       #sIntLoadUnloadOP(iStartSeqCond := (#sIntLoaderInSafePos AND #sMain.iStartSeqCond AND NOT #sIntLoadUnloadOP.sInterface.Error AND NOT "DB_LoaderShuttle2".sIntLoadUnloadOP.sInterface.SequenceRun AND #sIntLoadUnloadOP.sInterface.StartRequest AND #sShuttlePosInt),
                         iJobReq := #sIntLoadUnloadOP.sInterface.StartRequest,
                         iShuttleIntLoadUnloadPos := #tAxis_U_Position.IntLoadUnload,
                         iShuttleIntLoadUnloadPosSetPoint := "DB_AxisPosMachinePLC".Axis_U1.IntLoadUnload,
                         iShuttleIntLoadUnloadOP_Pos:=#tAxis_U_Position.IntLoadUnloadOP,
                         iShuttleIntLoadUnloadOP_PosSetPoint:="DB_AxisPosMachinePLC".Axis_U1.IntLoadUnloadOP,
                         iAxisV_LoadUnloadShuttlePos := #tAxis_V_Position.LoadUnload,
                         iAxisV_LoadUnloadShuttlePosSetPoint := "DB_AxisPosMachinePLC".Axis_V.Shuttle_1.LoadUnload,
                         iAxisV_SafePos := #tAxis_V_Position.Safe,
                         iAxisV_SafePosSetPoint := "DB_AxisPosMachinePLC".Axis_V.Safe,
                         iAxisW_SafePos := #tAxis_W_Position.Safe,
                         iAxisW_SafePosSetPoint := "DB_AxisPosMachinePLC".Axis_W.Safe,
                         iAxisW_ApproachLoadUnloadPos := #tAxis_W_Position.Approach,
                         iAxisW_ApproachLoadUnloadSetPoint := "DB_AxisPosMachinePLC".Axis_W.Shuttle_1.Approach,
                         iAxisW_LoadUnloadPos := #tAxis_W_Position.LoadUnload,
                         iAxisW_LoadUnloadPosSetPoint := "DB_AxisPosMachinePLC".Axis_W.Shuttle_1.LoadUnload,
                         iShuttleMoving := #iShuttleMoving,
                         iShuttleInPos := #iShuttleInPos,
                         iAxisV_Moving := #iAxisV_Moving,
                         iAxisV_InPos := #iAxisV_InPos,
                         iAxisW_Moving := #iAxisW_Moving,
                         iAxisW_InPos := #iAxisW_InPos,
                         iDrilledPartToUnload := "DB_PartManagement".sPosition.sGripper.Drilled.Presence.Part,
                         iUnDrilledPartToLoad := "DB_PartManagement".sPosition.sShuttle1.Undrilled.Presence.Part,
                         iLoadGripperClosed := #sIntLoadUnloadOP.iLoadGripperClosed,
                         iUnloadGripperOpen := "DB_GestionGripper".sDrilledGripper.oStateOpen,
                         iPLC_DateAndTime := "DB_ReadDateAndTime".sDateAndTime,
                         iStepPause := #sIntLoadUnloadOP.iStepPause,        
                         oShuttleStartReq => #sIntLoadUnloadOP.oShuttleStartReq,
                         oShuttlePosSetPoint => #sIntLoadUnloadOP.oShuttlePosSetPoint,
                         oAxisV_StartReq => #sIntLoadUnloadOP.oAxisV_StartReq,
                         oAxisV_PosSetPoint => #sIntLoadUnloadOP.oAxisV_PosSetPoint,
                         oAxisW_StartReq => #sIntLoadUnloadOP.oAxisW_StartReq,
                         oAxisW_PosSetPoint => #sIntLoadUnloadOP.oAxisW_PosSetPoint,
                         oLoadGripperCloseReq => #sIntLoadUnloadOP.oLoadGripperCloseReq,
                         oUnloadGripperOpenReq => #sIntLoadUnloadOP.oUnloadGripperOpenReq);
   END_REGION

   REGION Parts Control
       // Control In

       // Expected control result
      IF "DB_WorkingModes".sFilling THEN
          #sControlIn.iExpectedCtrlUndrilled := TRUE;
          #sControlIn.iExpectedCtrlDrilled := FALSE;
      ELSIF "DB_WorkingModes".sNormal THEN
          #sControlIn.iExpectedCtrlUndrilled := TRUE;
          #sControlIn.iExpectedCtrlDrilled := FALSE;
      ELSIF "DB_WorkingModes".sEmptying THEN
          #sControlIn.iExpectedCtrlUndrilled := FALSE;
          #sControlIn.iExpectedCtrlDrilled := FALSE;
      END_IF;

       #sControlIn(iStartSeqCond := (#sExtLoaderInSafePos AND #sMain.iStartSeqCond AND NOT #sControlIn.sInterface.Error AND NOT "DB_LoaderShuttle2".sControlIn.sInterface.SequenceRun AND #sControlIn.sInterface.StartRequest AND #sShuttlePosExt),
                   iJobReq := #sControlIn.sInterface.StartRequest,
                   iCtrlEnabled := TRUE,
                   iShuttleCtrlPos:= #tAxis_U_Position.PartControl,
                   iShuttleCtrlPosSetPoint:="DB_AxisPosMachinePLC".Axis_U1.PartControl,
                   iExpectedCtrlUndrilled := #sControlIn.iExpectedCtrlUndrilled,
                   iExpectedCtrlDrilled := #sControlIn.iExpectedCtrlDrilled,
                   iUndrilledPartPresence:= "DB_DigitalInputsBW_Station".sUndrilledPartCtrl.sSWStatus,
                   iDrilledPartPresence:= "DB_DigitalInputsBW_Station".sDrilledPartCtrl.sSWStatus,
                   iShuttleMoving := #iShuttleMoving,
                   iShuttleInPos := #iShuttleInPos,
                   iPLC_DateAndTime:= "DB_ReadDateAndTime".sDateAndTime,
                   iStepPause:=#sControlIn.iStepPause,       
                   oShuttleStartReq => #sControlIn.oShuttleStartReq,
                   oShuttlePosSetPoint => #sControlIn.oShuttlePosSetPoint,
                   oPartControlOK => #sControlIn.oPartControlOK,
                   oPartControlNOK => #sControlIn.oPartControlNOK);

       // Control Out

       // Expected control result
       #sControlOut.iExpectedCtrlUndrilled := "DB_PartManagement".sPosition.sShuttle1.Undrilled.Presence.Part;
       #sControlOut.iExpectedCtrlDrilled := "DB_PartManagement".sPosition.sShuttle1.Drilled.Presence.Part;

       #sControlOut(iStartSeqCond := (#sBwLoaderInSafePos AND #sMain.iStartSeqCond AND NOT #sControlOut.sInterface.Error AND NOT "DB_LoaderShuttle2".sControlOut.sInterface.SequenceRun AND #sControlOut.sInterface.StartRequest AND #sShuttlePosExt),
                    iJobReq := #sControlOut.sInterface.StartRequest,
                    iCtrlEnabled := TRUE,
                    iShuttleCtrlPos:= #tAxis_U_Position.PartControl,
                    iShuttleCtrlPosSetPoint:= "DB_AxisPosMachinePLC".Axis_U1.PartControl,
                    iExpectedCtrlUndrilled := #sControlOut.iExpectedCtrlUndrilled,
                    iExpectedCtrlDrilled := #sControlOut.iExpectedCtrlDrilled,
                    iUndrilledPartPresence:="DB_DigitalInputsBW_Station".sUndrilledPartCtrl.sSWStatus,
                    iDrilledPartPresence:="DB_DigitalInputsBW_Station".sDrilledPartCtrl.sSWStatus,
                    iShuttleMoving := #iShuttleMoving,
                    iShuttleInPos := #iShuttleInPos,
                    iPLC_DateAndTime:= "DB_ReadDateAndTime".sDateAndTime,
                    iStepPause:=#sControlOut.iStepPause,     
                    oShuttleStartReq => #sControlOut.oShuttleStartReq,
                    oShuttlePosSetPoint => #sControlOut.oShuttlePosSetPoint,
                    oPartControlOK => #sControlOut.oPartControlOK,
                    oPartControlNOK => #sControlOut.oPartControlNOK);
   END_REGION

   REGION BW Load Unload
       #sBwLoadUnload(iStartSeqCond:= (#sMain.iStartSeqCond AND NOT #sBwLoadUnload.sInterface.Error AND NOT "DB_LoaderShuttle2".sBwLoadUnload.sInterface.SequenceRun AND #sBwLoadUnload.sInterface.StartRequest AND #sShuttlePosExt),
                      iJobReq:= #sBwLoadUnload.sInterface.StartRequest,
                      iLoadReq:= #sMain.oBwLoadReq,
                      iUnloadReq:= #sMain.oBwUnloadReq,
                      iShuttleBwUnloadPos:= #tAxis_U_Position.BwUnload,
                      iShuttleBwUnloadPosSetPoint:= "DB_AxisPosMachinePLC".Axis_U1.BwUnLoad,
                      iShuttleBwLoadPos:= #tAxis_U_Position.BwLoad,
                      iShuttleBwLoadPosSetPoint:= "DB_AxisPosMachinePLC".Axis_U1.BwLoad,
                      iShuttleMoving:= #iShuttleMoving,
                      iShuttleInPos:= #iShuttleInPos,
                      iBwLoadDone:="DB_BwLoader".sBwCommunication.oLoadJobDone,
                      iBwUnloadDone:="DB_BwLoader".sBwCommunication.oUnloadJobDone,
                      iBwLoaderInSafePos:=#sBwLoaderInSafePos,
                      iPLC_DateAndTime:= "DB_ReadDateAndTime".sDateAndTime,
                      iStepPause:=#sBwLoadUnload.iStepPause,      
                      oShuttleStartReq=> #sBwLoadUnload.oShuttleStartReq,
                      oShuttlePosSetPoint=> #sBwLoadUnload.oShuttlePosSetPoint,
                      oBwLoadReq=> #sBwLoadUnload.oBwLoadReq,
                      oBwUnloadReq=>#sBwLoadUnload.oBwUnloadReq);
   END_REGION

   REGION BW Control
       // BW Control In

       // Expected control result
       #sBwControlIn.iExpectedCtrl := "DB_PartManagement".sPosition.sShuttle1.Undrilled.Presence.Part;

       #sBwControlIn(iStartSeqCond := (#sMain.iStartSeqCond AND NOT #sBwControlIn.sInterface.Error AND NOT "DB_LoaderShuttle2".sBwControlIn.sInterface.SequenceRun AND #sBwControlIn.sInterface.StartRequest AND #sShuttlePosExt),
                     iJobReq := #sBwControlIn.sInterface.StartRequest,
                     iCtrlEnabled := TRUE,
                     iShuttleCtrlPos := #tAxis_U_Position.BwControl,
                     iShuttleCtrlPosSetPoint := "DB_AxisPosMachinePLC".Axis_U1.BwControl,
                     iExpectedCtrl := #sBwControlIn.iExpectedCtrl,
                     iBwPresence := "DB_DigitalInputsBW_Station".sBwCtrl.sSWStatus,
                     iShuttleMoving := #iShuttleMoving,
                     iShuttleInPos := #iShuttleInPos,
                     iPLC_DateAndTime := "DB_ReadDateAndTime".sDateAndTime,
                     iStepPause := #sBwControlIn.iStepPause,     
                     oShuttleStartReq => #sBwControlIn.oShuttleStartReq,
                     oShuttlePosSetPoint => #sBwControlIn.oShuttlePosSetPoint,
                     oBwControlOK => #sBwControlIn.oBwControlOK,
                     oBwControlNOK => #sBwControlIn.oBwControlNOK);

       #sBwConsecutiveCtrl(iReset:=#sBwConsecutiveCtrl.oConsecutiveError AND #sActBwControlIn.sCurrent_Step_NB = 60,
                           iGoodEntry:=#sBwControlIn.oBwControlOK,
                           iBadEntry:=#sBwControlIn.oBwControlNOK,
                           iPresetValue:=3,
                           oConsecutiveError=>#sBwConsecutiveCtrl.oConsecutiveError);
   END_REGION

   REGION Blowing
       #sBlowing(iStartSeqCond:=(#sIntLoaderInSafePos AND #sMain.iStartSeqCond AND NOT #sBlowing.sInterface.Error AND NOT "DB_LoaderShuttle2".sBlowing.sInterface.SequenceRun AND #sBlowing.sInterface.StartRequest AND #sShuttlePosInt),
                 iJobReq:=#sBlowing.sInterface.StartRequest,
                 iShuttleBlowingPos:=#tAxis_U_Position.Blowing,
                 iShuttleBlowingPosSetPoint:="DB_AxisPosMachinePLC".Axis_U1.Blowing,
                 iAxisV_BlowingPos:=#tAxis_V_Position.Blowing,
                 iAxisV_BlowingPosSetPoint:="DB_AxisPosMachinePLC".Axis_V.Shuttle_1.Blowing,
                 iAxisW_SafePos:=#tAxis_W_Position.Safe,
                 iAxisW_SafePosSetPoint:="DB_AxisPosMachinePLC".Axis_W.Safe,
                 iAxisW_BlowingPos:=#tAxis_W_Position.Blowing,
                 iAxisW_BlowingPosSetPoint:="DB_AxisPosMachinePLC".Axis_W.Shuttle_1.Blowing,
                 iShuttleMoving:=#iShuttleMoving,
                 iShuttleInPos:=#iShuttleInPos,
                 iAxisV_Moving:=#iAxisV_Moving,
                 iAxisV_InPos:=#iAxisV_InPos,
                 iAxisW_Moving:=#iAxisW_Moving,
                 iAxisW_InPos:=#iAxisW_InPos,
                 iBlowingTime:=DINT_TO_TIME(REAL_TO_DINT("DB_HMISetting".BlowingSetpoint)),
                 iPLC_DateAndTime:="DB_ReadDateAndTime".sDateAndTime,
                 iStepPause:=#sBlowing.iStepPause,
                 oShuttleStartReq=>#sBlowing.oShuttleStartReq,
                 oShuttlePosSetPoint=>#sBlowing.oShuttlePosSetPoint,
                 oAxisV_StartReq=>#sBlowing.oAxisV_StartReq,
                 oAxisV_PosSetPoint=>#sBlowing.iAxisV_BlowingPosSetPoint,
                 oAxisW_StartReq=>#sBlowing.oAxisW_StartReq,
                 oAxisW_PosSetPoint=>#sBlowing.iAxisW_BlowingPosSetPoint,
                 oBlowingReq=>#sBlowing.oBlowingReq);
   END_REGION

   REGION Action Part Control In
       // Conditions d'arrêt en Mode Auto
       #sActPartControlIn.iModeAutoPosCondition :=
          ("DB_WorkingModes".sAuto AND (#sControlIn.sMissingPartCtrlUndrilled OR #sControlIn.sMissingPartCtrlDrilled) AND "DB_LoaderOptions".ActPartControlIn.Stop)
       OR ("DB_WorkingModes".sAuto AND (#sControlIn.sExtraPartCtrlUndrilled OR #sControlIn.sExtraPartCtrlDrilled) AND "DB_LoaderOptions".ActPartControlIn.Stop)
       OR ("DB_WorkingModes".sAuto AND (#sControlIn.sExtraPartCtrlUndrilled OR #sControlIn.sExtraPartCtrlDrilled) AND NOT "DB_LoaderOptions".ActPartControlIn.Stop);
       // Conditions d'arrêt en Mode Semi Auto   
       #sActPartControlIn.iModeSemiAutoPosCondition :=
          ("DB_WorkingModes".sSemiAuto AND (#sControlIn.sMissingPartCtrlUndrilled OR #sControlIn.sMissingPartCtrlDrilled) AND "DB_LoaderOptions".ActPartControlIn.Stop)
       OR ("DB_WorkingModes".sSemiAuto AND (#sControlIn.sExtraPartCtrlUndrilled OR #sControlIn.sExtraPartCtrlDrilled) AND "DB_LoaderOptions".ActPartControlIn.Stop)
       OR ("DB_WorkingModes".sSemiAuto AND (#sControlIn.sExtraPartCtrlUndrilled OR #sControlIn.sExtraPartCtrlDrilled) AND NOT "DB_LoaderOptions".ActPartControlIn.Stop);
       // Conditions pas d'arrêt
       #sActPartControlIn.iNoStopCondition :=
          ("DB_WorkingModes".sAuto AND (#sControlIn.sMissingPartCtrlUndrilled OR #sControlIn.sMissingPartCtrlDrilled) AND NOT "DB_LoaderOptions".ActPartControlIn.Stop)
       OR ("DB_WorkingModes".sSemiAuto AND (#sControlIn.sMissingPartCtrlUndrilled OR #sControlIn.sMissingPartCtrlDrilled) AND NOT "DB_LoaderOptions".ActPartControlIn.Stop);

       #sActPartControlIn(iStartSeqCond:= (#sMain.iStartSeqCond AND NOT #sActPartControlIn.sInterface.Error AND NOT "DB_LoaderShuttle2".sActPartControlIn.sInterface.SequenceRun AND #sActPartControlIn.sInterface.StartRequest AND #sShuttlePosExt),
                          iJobReq:= #sActPartControlIn.sInterface.StartRequest,
                          iShuttleModeAutoPos:= #tAxis_U_Position.ExtLoadUnloadAuto,
                          iShuttleModeAutoPosSetPoint:= "DB_AxisPosMachinePLC".Axis_U1.ExtLoadUnloadAuto,
                          iShuttleModeSemiAutoPos:= #tAxis_U_Position.ExtLoadUnloadManu,
                          iShuttleModeSemiAutoPosSetPoint:= "DB_AxisPosMachinePLC".Axis_U1.ExtLoadUnloadManu,
                          iShuttleMoving:= #iShuttleMoving,
                          iShuttleInPos:= #iShuttleInPos,
                          iModeAutoPosCondition:= #sActPartControlIn.iModeAutoPosCondition,
                          iModeSemiAutoPosCondition:= #sActPartControlIn.iModeSemiAutoPosCondition,
                          iNoStopCondition:= #sActPartControlIn.iNoStopCondition,
                          iOperatorCycleRestart:= "LBP_Chan1".E_ProgRunning,
                          iNC_Stopped:= NOT "LBP_Chan1".E_ProgRunning,
                          iNC_Running:= "LBP_Chan1".E_ProgRunning,
                          iMissingPart:=#sControlIn.sMissingPartCtrlUndrilled OR #sControlIn.sMissingPartCtrlDrilled,
                          iExtraPart:=#sControlIn.sExtraPartCtrlUndrilled OR #sControlIn.sExtraPartCtrlDrilled,
                          iPLC_DateAndTime:= "DB_ReadDateAndTime".sDateAndTime,
                          iStepPause:= #sActPartControlIn.iStepPause,
                          oShuttleStartReq=> #sActPartControlIn.oShuttleStartReq,
                          oShuttlePosSetPoint=> #sActPartControlIn.oShuttlePosSetPoint,
                          oStopNC_Req=> #sActPartControlIn.oStopNC_Req,       // Implicite par Alarm Message
                          oRestartNC_Req=> #sActPartControlIn.oRestartNC_Req, // Implicite par Restart NC
                          oRestartStep=> #sActPartControlIn.oRestartStep,
                          oContinuationStep=> #sActPartControlIn.oContinuationStep,
                          oMsgMissingPart=>#sActPartControlIn.oMsgMissingPart,
                          oMsgExtraPart=>#sActPartControlIn.oMsgExtraPart);

       #sRT_PartControlInMissing(CLK := #sActPartControlIn.oMsgMissingPart);
       IF #sRT_PartControlInMissing.Q THEN
           "LBP_AlarmMsgs".UserA[03].A70UUxx[15] := TRUE;
       END_IF;

       #sRT_PartControlInExtra(CLK := #sActPartControlIn.oMsgExtraPart);
       IF #sRT_PartControlInExtra.Q THEN
           "LBP_AlarmMsgs".UserA[03].A70UUxx[16] := TRUE;
       END_IF;
   END_REGION

   REGION Action Part Control Out
       // Conditions d'arrêt en Mode Auto
       #sActPartControlOut.iModeAutoPosCondition :=
          ("DB_WorkingModes".sAuto AND (#sControlOut.sMissingPartCtrlUndrilled OR #sControlOut.sMissingPartCtrlDrilled) AND "DB_LoaderOptions".ActPartControlOut.Stop)
       OR ("DB_WorkingModes".sAuto AND (#sControlOut.sExtraPartCtrlUndrilled OR #sControlOut.sExtraPartCtrlDrilled) AND "DB_LoaderOptions".ActPartControlOut.Stop)
       OR ("DB_WorkingModes".sAuto AND (#sControlOut.sExtraPartCtrlUndrilled OR #sControlOut.sExtraPartCtrlDrilled) AND NOT "DB_LoaderOptions".ActPartControlOut.Stop);
       // Conditions d'arrêt en Mode Semi Auto 
       #sActPartControlOut.iModeSemiAutoPosCondition :=
          ("DB_WorkingModes".sSemiAuto AND (#sControlOut.sMissingPartCtrlUndrilled OR #sControlOut.sMissingPartCtrlDrilled) AND "DB_LoaderOptions".ActPartControlOut.Stop)
       OR ("DB_WorkingModes".sSemiAuto AND (#sControlOut.sExtraPartCtrlUndrilled OR #sControlOut.sExtraPartCtrlDrilled) AND "DB_LoaderOptions".ActPartControlOut.Stop)
       OR ("DB_WorkingModes".sSemiAuto AND (#sControlOut.sExtraPartCtrlUndrilled OR #sControlOut.sExtraPartCtrlDrilled) AND NOT "DB_LoaderOptions".ActPartControlOut.Stop);
       // Conditions pas d'arrêt
       #sActPartControlOut.iNoStopCondition :=
          ("DB_WorkingModes".sAuto AND (#sControlOut.sMissingPartCtrlUndrilled OR #sControlOut.sMissingPartCtrlDrilled) AND NOT "DB_LoaderOptions".ActPartControlOut.Stop)
       OR ("DB_WorkingModes".sSemiAuto AND (#sControlOut.sMissingPartCtrlUndrilled OR #sControlOut.sMissingPartCtrlDrilled) AND NOT "DB_LoaderOptions".ActPartControlOut.Stop);

       #sActPartControlOut(iStartSeqCond := (#sMain.iStartSeqCond AND NOT #sActPartControlOut.sInterface.Error AND NOT "DB_LoaderShuttle2".sActPartControlout.sInterface.SequenceRun AND #sActPartControlOut.sInterface.StartRequest AND #sShuttlePosExt),
                           iJobReq := #sActPartControlOut.sInterface.StartRequest,
                           iShuttleModeAutoPos := #tAxis_U_Position.ExtLoadUnloadAuto,
                           iShuttleModeAutoPosSetPoint := "DB_AxisPosMachinePLC".Axis_U1.ExtLoadUnloadAuto,
                           iShuttleModeSemiAutoPos := #tAxis_U_Position.ExtLoadUnloadManu,
                           iShuttleModeSemiAutoPosSetPoint := "DB_AxisPosMachinePLC".Axis_U1.ExtLoadUnloadManu,
                           iShuttleMoving := #iShuttleMoving,
                           iShuttleInPos := #iShuttleInPos,
                           iModeAutoPosCondition := #sActPartControlOut.iModeAutoPosCondition,
                           iModeSemiAutoPosCondition := #sActPartControlOut.iModeSemiAutoPosCondition,
                           iNoStopCondition:=#sActPartControlOut.iNoStopCondition,
                           iOperatorCycleRestart := "LBP_Chan1".E_ProgRunning,
                           iNC_Stopped := NOT "LBP_Chan1".E_ProgRunning,
                           iNC_Running := "LBP_Chan1".E_ProgRunning,
                           iMissingPart:=#sControlOut.sMissingPartCtrlUndrilled OR #sControlOut.sMissingPartCtrlDrilled,
                           iExtraPart:=#sControlOut.sExtraPartCtrlUndrilled OR #sControlOut.sExtraPartCtrlDrilled,
                           iPLC_DateAndTime := "DB_ReadDateAndTime".sDateAndTime,
                           iStepPause := #sActPartControlOut.iStepPause, 
                           oShuttleStartReq => #sActPartControlOut.oShuttleStartReq,
                           oShuttlePosSetPoint => #sActPartControlOut.oShuttlePosSetPoint,
                           oStopNC_Req => #sActPartControlOut.oStopNC_Req,       // Implicite par Alarm Message
                           oRestartNC_Req => #sActPartControlOut.oRestartNC_Req, // Implicite par Restart NC
                           oRestartStep => #sActPartControlOut.oRestartStep,
                           oContinuationStep => #sActPartControlOut.oContinuationStep,
                           oMsgMissingPart=>#sActPartControlOut.oMsgMissingPart,
                           oMsgExtraPart=>#sActPartControlOut.oMsgExtraPart);

      #sRT_PartControlOutMissing(CLK := #sActPartControlOut.oMsgMissingPart);
      IF #sRT_PartControlOutMissing.Q THEN
          "LBP_AlarmMsgs".UserA[03].A70UUxx[17] := TRUE;
      END_IF;

      #sRT_PartControlOutExtra(CLK := #sActPartControlOut.oMsgExtraPart);
      IF #sRT_PartControlOutExtra.Q THEN
          "LBP_AlarmMsgs".UserA[03].A70UUxx[18] := TRUE;
      END_IF;
   END_REGION

   REGION Action Bw Control In
       // Conditions d'arrêt en Mode Auto
       #sActBwControlIn.iModeAutoPosCondition :=
       ("DB_WorkingModes".sAuto AND #sBwControlIn.sMissingBwCtrl AND ("DB_LoaderOptions".ActBwControlIn.Stop OR #sBwConsecutiveCtrl.oConsecutiveError))
       OR ("DB_WorkingModes".sAuto AND #sBwControlIn.sExtraBwCtrl AND "DB_LoaderOptions".ActBwControlIn.Stop)
       OR ("DB_WorkingModes".sAuto AND #sBwControlIn.sExtraBwCtrl AND NOT "DB_LoaderOptions".ActBwControlIn.Stop);
       // Conditions d'arrêt en Mode Semi Auto
       #sActBwControlIn.iModeSemiAutoPosCondition :=
          ("DB_WorkingModes".sSemiAuto AND #sBwControlIn.sMissingBwCtrl AND "DB_LoaderOptions".ActBwControlIn.Stop)
       OR ("DB_WorkingModes".sSemiAuto AND #sBwControlIn.sExtraBwCtrl AND "DB_LoaderOptions".ActBwControlIn.Stop)
       OR ("DB_WorkingModes".sSemiAuto AND #sBwControlIn.sExtraBwCtrl AND NOT "DB_LoaderOptions".ActBwControlIn.Stop);
       // Conditions pas d'arrêt
       #sActBwControlIn.iNoStopCondition :=
       ("DB_WorkingModes".sAuto AND #sBwControlIn.sMissingBwCtrl AND (NOT "DB_LoaderOptions".ActBwControlIn.Stop AND NOT #sBwConsecutiveCtrl.oConsecutiveError))
       OR ("DB_WorkingModes".sSemiAuto AND #sBwControlIn.sMissingBwCtrl AND NOT "DB_LoaderOptions".ActBwControlIn.Stop);

       #sActBwControlIn(iStartSeqCond := (#sMain.iStartSeqCond AND NOT #sActBwControlIn.sInterface.Error AND NOT "DB_LoaderShuttle2".sActBwControlIn.sInterface.SequenceRun AND #sActBwControlIn.sInterface.StartRequest AND #sShuttlePosExt),
                        iJobReq := #sActBwControlIn.sInterface.StartRequest,
                        iShuttleModeAutoPos := #tAxis_U_Position.BwLoad,
                        iShuttleModeAutoPosSetPoint := "DB_AxisPosMachinePLC".Axis_U1.BwLoad,
                        iShuttleModeSemiAutoPos := #tAxis_U_Position.BwLoad,
                        iShuttleModeSemiAutoPosSetPoint := "DB_AxisPosMachinePLC".Axis_U1.BwLoad,
                        iShuttleMoving := #iShuttleMoving,
                        iShuttleInPos := #iShuttleInPos,
                        iModeAutoPosCondition := #sActBwControlIn.iModeAutoPosCondition,
                        iModeSemiAutoPosCondition := #sActBwControlIn.iModeSemiAutoPosCondition,
                        iNoStopCondition:=#sActBwControlIn.iNoStopCondition,
                        iOperatorCycleRestart := "LBP_Chan1".E_ProgRunning,
                        iNC_Stopped :=  (NOT "LBP_Chan1".E_ProgRunning AND "DB_OPC_Machine".Parameters.ConsecutiveBwIn = 0) OR "DB_OPC_Machine".Parameters.ConsecutiveBwIn > 0,
                        iNC_Running := "LBP_Chan1".E_ProgRunning,
                        iMissingPart:=#sBwControlIn.sMissingBwCtrl,
                        iExtraPart:=#sBwControlIn.sExtraBwCtrl,
                        iPLC_DateAndTime := "DB_ReadDateAndTime".sDateAndTime,
                        iStepPause := #sActBwControlIn.iStepPause,
                        oShuttleStartReq => #sActBwControlIn.oShuttleStartReq,
                        oShuttlePosSetPoint => #sActBwControlIn.oShuttlePosSetPoint,
                        oStopNC_Req => #sActBwControlIn.oStopNC_Req,       // Implicite par Alarm Message
                        oRestartNC_Req => #sActBwControlIn.oRestartNC_Req, // Implicite par Restart NC
                        oRestartStep => #sActBwControlIn.oRestartStep,
                        oContinuationStep => #sActBwControlIn.oContinuationStep,
                        oMsgMissingPart=>#sActBwControlIn.oMsgMissingPart,
                        oMsgExtraPart=>#sActBwControlIn.iExtraPart);

       IF "DB_OPC_Machine".Parameters.ConsecutiveBwIn = 0 THEN
           #sRT_BwControlInMissing(CLK := #sActBwControlIn.oMsgMissingPart);
           IF #sRT_BwControlInMissing.Q THEN
               "LBP_AlarmMsgs".UserA[03].A70UUxx[19] := TRUE;
           END_IF;

           #sRT_BwControlInExtra(CLK := #sActBwControlIn.iExtraPart);
           IF #sRT_BwControlInExtra.Q THEN
               "LBP_AlarmMsgs".UserA[03].A70UUxx[20] := TRUE;
           END_IF;
       ELSE
           "LBP_AlarmMsgs".UserA[03].A70UUxx[19] := FALSE;
           "LBP_AlarmMsgs".UserA[03].A70UUxx[20] := FALSE;
       END_IF;
   END_REGION

   REGION Axis U-V-W Start Request
       // Axis U - Start Request
       #oShuttleStartReq :=
       #sShuttleInt.oShuttleStartReq
       OR #sShuttleExt.oShuttleStartReq
       OR #sControlIn.oShuttleStartReq
       OR #sControlOut.oShuttleStartReq
       OR #sBlowing.oShuttleStartReq
       OR #sIntLoadUnload.oShuttleStartReq
       OR #sIntLoadUnloadOP.oShuttleStartReq
       OR #sExtLoadUnload.oShuttleStartReq
       OR #sBwLoadUnload.oShuttleStartReq
       OR #sBwControlIn.oShuttleStartReq
       OR #sActPartControlIn.oShuttleStartReq
       OR #sActPartControlOut.oShuttleStartReq
       OR #sActBwControlIn.oShuttleStartReq;

       // Axis U - Position Set point according to start request
       IF #sShuttleInt.oShuttleStartReq THEN
           #oShuttlePosSetPoint := #sShuttleInt.oShuttlePosSetPoint;
       ELSIF #sShuttleExt.oShuttleStartReq THEN
           #oShuttlePosSetPoint := #sShuttleExt.oShuttlePosSetPoint;
       ELSIF #sControlIn.oShuttleStartReq THEN
           #oShuttlePosSetPoint := #sControlIn.oShuttlePosSetPoint;
       ELSIF #sControlOut.oShuttleStartReq THEN
           #oShuttlePosSetPoint := #sControlOut.oShuttlePosSetPoint;
       ELSIF #sExtLoadUnload.oShuttleStartReq THEN
           #oShuttlePosSetPoint := #sExtLoadUnload.oShuttlePosSetPoint;
       ELSIF #sIntLoadUnload.oShuttleStartReq THEN
           #oShuttlePosSetPoint := #sIntLoadUnload.oShuttlePosSetPoint;
       ELSIF #sIntLoadUnloadOP.oShuttleStartReq THEN
           #oShuttlePosSetPoint := #sIntLoadUnloadOP.oShuttlePosSetPoint;
       ELSIF #sBwLoadUnload.oShuttleStartReq THEN
           #oShuttlePosSetPoint := #sBwLoadUnload.oShuttlePosSetPoint;
       ELSIF #sBwControlIn.oShuttleStartReq THEN
           #oShuttlePosSetPoint := #sBwControlIn.oShuttlePosSetPoint;
       ELSIF #sActPartControlIn.oShuttleStartReq THEN
           #oShuttlePosSetPoint := #sActPartControlIn.oShuttlePosSetPoint;
       ELSIF #sActPartControlOut.oShuttleStartReq THEN
           #oShuttlePosSetPoint := #sActPartControlOut.oShuttlePosSetPoint;
       ELSIF #sActBwControlIn.oShuttleStartReq THEN
           #oShuttlePosSetPoint := #sActBwControlIn.oShuttlePosSetPoint;
       ELSIF #sBlowing.oShuttleStartReq THEN
           #oShuttlePosSetPoint := #sBlowing.oShuttlePosSetPoint;
       ELSE
           #oShuttleStartReq := FALSE;
       END_IF;

       // Axis V - Start Request
       #oAxisVStartReq :=
       #sIntLoadUnload.oAxisV_StartReq
       OR #sIntLoadUnloadOP.oAxisV_StartReq
       OR #sBlowing.oAxisV_StartReq;

       // Axis V - Position Set point  according to start request
       IF #sIntLoadUnload.oAxisV_StartReq THEN
           #oAxisVPosSetPoint := #sIntLoadUnload.oAxisV_PosSetPoint;
       ELSIF #sIntLoadUnloadOP.oAxisV_StartReq THEN
           #oAxisVPosSetPoint := #sIntLoadUnloadOP.oAxisV_PosSetPoint;
       ELSIF #sBlowing.oAxisV_StartReq THEN
           #oAxisVPosSetPoint := #sBlowing.oAxisV_PosSetPoint;
       ELSE
           #oAxisVStartReq := FALSE;
       END_IF;

       // Axis W - Start Request
       #oAxisWStartReq :=
       #sIntLoadUnload.oAxisW_StartReq
       OR #sIntLoadUnloadOP.oAxisW_StartReq
       OR #sBlowing.oAxisW_StartReq;

       // Axis W - Position Set point  according to start request
       IF #sIntLoadUnload.oAxisW_StartReq THEN
           #oAxisWPosSetPoint := #sIntLoadUnload.oAxisW_PosSetPoint;
       ELSIF #sIntLoadUnloadOP.oAxisW_StartReq THEN
           #oAxisWPosSetPoint := #sIntLoadUnloadOP.oAxisW_PosSetPoint;
       ELSIF #sBlowing.oAxisW_StartReq THEN
           #oAxisWPosSetPoint := #sBlowing.oAxisW_PosSetPoint;
       ELSE
           #oAxisWStartReq := FALSE;
       END_IF;
   END_REGION

   REGION Gates Command Request
       // External Gate
       #oExtGateOpenReq := #sShuttleInt.oExtGateOpenReq OR #sShuttleExt.oExtGateOpenReq;
       #oExtGateCloseReq := #sShuttleInt.oExtGateCloseReq OR #sShuttleExt.oExtGateCloseReq;

       // Internal Gate
       #oIntGateOpenReq := #sShuttleInt.oIntGateOpenReq OR #sShuttleExt.oIntGateOpenReq;
       #oIntGateCloseReq := #sShuttleInt.oIntGateCloseReq OR #sShuttleExt.oIntGateCloseReq;
   END_REGION

   REGION Gripper Command Request
       // Load Gripper
       #oLoadGripperCloseReq := #sIntLoadUnload.oLoadGripperCloseReq
       OR #sIntLoadUnloadOP.oLoadGripperCloseReq;
       // Unload Gripper
       #oUnloadGripperOpenReq := #sIntLoadUnload.oUnloadGripperOpenReq
       OR #sIntLoadUnloadOP.oUnloadGripperOpenReq;
   END_REGION

   REGION Blowing Command Request
       #oBlowingReq := #sBlowing.oBlowingReq;
   END_REGION
END_FUNCTION_BLOCK

FUNCTION_BLOCK "FB_Main"   // FB69, SCL
{ S7_Optimized_Access := 'TRUE' }
// stored: MemoryReserve 100, SetENOAutomatically false
   VAR_INPUT
      iStartSeqCond : Bool;
      iJobReq : Bool;
      iShuttleINT : Bool;
      iShuttleSAS : Bool;
      iShuttleEXT : Bool;
      iGripperReserved : Bool;
      iGripperReleased : Bool;
      iShuttleUndrilledPart : Bool;
      iShuttleDrilledPart : Bool;
      iShuttleUndrilledBw : Bool;
      iShuttleDrilledBw : Bool;
      iPartCtrlInOK : Bool;
      iPartCtrlInNOK : Bool;
      iPartCtrlInContinuationStep : Bool;
      iPartCtrlInRestartStep : Bool;
      iPartCtrlOutOK : Bool;
      iPartCtrlOutNOK : Bool;
      iPartCtrlOutContinuationStep : Bool;
      iPartCtrlOutRestartStep : Bool;
      iBwCtrlInOK : Bool;
      iBwCtrlInNOK : Bool;
      iBwCtrlInContinuationStep : Bool;
      iBwCtrlInRestartStep : Bool;
      iGripperOK : Bool;
      iNC_NoNeedAxis : Bool;
      iExtLoaderInSafePos : Bool;
      iIntLoaderInSafePos : Bool;
      iBwLoaderInSafePos : Bool;
      iOnePieceMode : Bool;
      iPLC_DateAndTime : DTL;
      iStepPause : Bool;
   END_VAR
   VAR_OUTPUT
      oGripperAxisRequest : Bool;
      oGripperAxisRelease : Bool;
      oNoExtLoad : Bool;
      oBwLoadReq : Bool;
      oBwUnloadReq : Bool;
   END_VAR
   VAR_IN_OUT
      ioShuttleIntSeq : "UDT_SequenceInterface";
      ioShuttleExtSeq : "UDT_SequenceInterface";
      ioControlInSeq : "UDT_SequenceInterface";
      ioControlOutSeq : "UDT_SequenceInterface";
      ioBlowingSeq : "UDT_SequenceInterface";
      ioIntLoadUnloadSeq : "UDT_SequenceInterface";
      ioIntLoadUnloadOP_Seq : "UDT_SequenceInterface";
      ioExtLoadUnloadSeq : "UDT_SequenceInterface";
      ioBWLoadUnloadSeq : "UDT_SequenceInterface";
      ioBWControlSeq : "UDT_SequenceInterface";
      ioActPartControlInSeq : "UDT_SequenceInterface";
      ioActPartControlOutSeq : "UDT_SequenceInterface";
      ioActBwControlInSeq : "UDT_SequenceInterface";
   END_VAR
   VAR
      sCurrent_Step_NB : Int;   // Active Step Number
      sCheck_Step_Condition : Bool;
      sOneStepForward : Bool;
      sRTOneStepForward : R_TRIG;
      sOneStepMode { S7_SetPoint := 'True'} : Bool;
      sStepForward : Bool;
      sInterface : "UDT_SequenceInterface";
      sGripperAxisRequest : Bool;
      sGripperAxisRelease : Bool;
      sHistory : Struct
         Activation : Bool;
         Steps : Array[0..99] of Int;
         Date_Time : Array[0..99] of DTL;
      END_STRUCT;
      StepText : "FB_GetTextErrorCode";
   END_VAR
   VAR_TEMP
      tIndex : Int;   // Index
   END_VAR
   VAR CONSTANT
      S00_INIT_STEP : Int := 0;
      S10_SHUTTLE_EXT_SEQ_REQUEST : Int := 10;
      S12_SHUTTLE_EXT_SEQ_IN_PROGRESS : Int := 12;
      S14_SHUTTLE_EXT_SEQ_ACQUIT : Int := 14;
      S19_SHUTTLE_EXT_SEQ_ERROR : Int := 19;
      S20_EXT_LOAD_UNLOAD_SEQ_REQUEST : Int := 20;
      S22_EXT_LOAD_UNLOAD_SEQ_IN_PROGRESS : Int := 22;
      S24_EXT_LOAD_UNLOAD_SEQ_ACQUIT : Int := 24;
      S29_EXT_LOAD_UNLOAD_SEQ_ERROR : Int := 29;
      S30_PARTS_CTRL_IN_SEQ_REQUEST : Int := 30;
      S32_PARTS_CTRL_IN_SEQ_IN_PROGRESS : Int := 32;
      S34_PARTS_CTRL_IN_SEQ_ACQUIT : Int := 34;
      S39_PARTS_CTRL_IN_SEQ_ERROR : Int := 39;
      S40_BW_LOAD_UNLOAD_SEQ_REQUEST : Int := 40;
      S42_BW_LOAD_UNLOAD_SEQ_IN_PROGRESS : Int := 42;
      S44_BW_LOAD_UNLOAD_SEQ_ACQUIT : Int := 44;
      S49_BW_LOAD_UNLOAD_SEQ_ERROR : Int := 49;
      S50_BW_CTRL_UNLOAD_SEQ_REQUEST : Int := 50;
      S52_BW_CTRL_UNLOAD_SEQ_IN_PROGRESS : Int := 52;
      S54_BW_CTRL_UNLOAD_SEQ_ACQUIT : Int := 54;
      S59_BW_CTRL_UNLOAD_SEQ_ERROR : Int := 59;
      S60_SHUTTLE_INT_SEQ_REQUEST : Int := 60;
      S62_SHUTTLE_INT_SEQ_IN_PROGRESS : Int := 62;
      S64_SHUTTLE_INT_SEQ_ACQUIT : Int := 64;
      S69_SHUTTLE_INT_SEQ_ERROR : Int := 69;
      S70_TRANSFER_V_AND_W_AXIS_TO_PLC : Int := 70;
      S80_INT_LOAD_UNLOAD_SEQ_REQUEST : Int := 80;
      S82_INT_LOAD_UNLOAD_SEQ_IN_PROGRESS : Int := 82;
      S84_INT_LOAD_UNLOAD_SEQ_ACQUIT : Int := 84;
      S89_INT_LOAD_UNLOAD_SEQ_ERROR : Int := 89;
      S90_TRANSFER_V_AND_W_AXIS_TO_NC : Int := 90;
      S100_SHUTTLE_EXT_SEQ_REQUEST : Int := 100;
      S102_SHUTTLE_EXT_SEQ_IN_PROGRESS : Int := 102;
      S104_SHUTTLE_EXT_SEQ_ACQUIT : Int := 104;
      S109_SHUTTLE_EXT_SEQ_ERROR : Int := 109;
      S110_BW_LOAD_UNLOAD_SEQ_REQUEST : Int := 110;
      S112_BW_LOAD_UNLOAD_SEQ_IN_PROGRESS : Int := 112;
      S114_BW_LOAD_UNLOAD_SEQ_ACQUIT : Int := 114;
      S119_BW_LOAD_UNLOAD_SEQ_ERROR : Int := 119;
      S120_PARTS_CTRL_OUT_SEQ_REQUEST : Int := 120;
      S122_PARTS_CTRL_OUT_SEQ_IN_PROGRESS : Int := 122;
      S124_PARTS_CTRL_OUT_SEQ_ACQUIT : Int := 124;
      S129_PARTS_CTRL_OUT_SEQ_ERROR : Int := 129;
      S130_CHECK_CYCLE_STOP : Int := 130;
      S140_EXT_LOAD_UNLOAD_SEQ_REQUEST : Int := 140;
      S142_EXT_LOAD_UNLOAD_SEQ_IN_PROGRESS : Int := 142;
      S144_EXT_LOAD_UNLOAD_SEQ_ACQUIT : Int := 144;
      S149_EXT_LOAD_UNLOAD_SEQ_ERROR : Int := 149;
      S200_BLOWING_SEQ_REQUEST : Int := 200;
      S202_BLOWING_SEQ_IN_PROGRESS : Int := 202;
      S204_BLOWING_SEQ_ACQUIT : Int := 204;
      S209_BLOWING_SEQ_ERROR : Int := 209;
      S210_INT_LOAD_UNLOAD_OP_SEQ_REQUEST : Int := 210;
      S212_INT_LOAD_UNLOAD_OP_SEQ_IN_PROGRESS : Int := 212;
      S214_INT_LOAD_UNLOAD_OP_SEQ_ACQUIT : Int := 214;
      S219_INT_LOAD_UNLOAD_OP_SEQ_ERROR : Int := 219;
      S300_ACT_PART_CTRL_IN_SEQ_REQUEST : Int := 300;
      S302_ACT_PART_CTRL_IN_SEQ_IN_PROGRESS : Int := 302;
      S304_ACT_PART_CTRL_IN_SEQ_ACQUIT : Int := 304;
      S309_ACT_PART_CTRL_IN_SEQ_ERROR : Int := 309;
      S310_ACT_PART_CTRL_OUT_SEQ_REQUEST : Int := 310;
      S312_ACT_PART_CTRL_OUT_SEQ_IN_PROGRESS : Int := 312;
      S314_ACT_PART_CTRL_OUT_SEQ_ACQUIT : Int := 314;
      S319_ACT_PART_CTRL_OUT_SEQ_ERROR : Int := 319;
      S320_ACT_BW_CTRL_IN_SEQ_REQUEST : Int := 320;
      S322_ACT_BW_CTRL_IN_SEQ_IN_PROGRESS : Int := 322;
      S324_ACT_BW_CTRL_IN_SEQ_ACQUIT : Int := 324;
      S329_ACT_BW_CTRL_IN_SEQ_ERROR : Int := 329;
      S999_ERROR : Int := 999;
   END_VAR
   // StepText.sCode_error[0].ErrorCode := 0;
   // StepText.sCode_error[1].ErrorCode := 12;
   // StepText.sCode_error[2].ErrorCode := 22;
   // StepText.sCode_error[3].ErrorCode := 32;
   // StepText.sCode_error[4].ErrorCode := 42;
   // StepText.sCode_error[5].ErrorCode := 52;
   // StepText.sCode_error[6].ErrorCode := 62;
   // StepText.sCode_error[7].ErrorCode := 82;
   // StepText.sCode_error[8].ErrorCode := 102;
   // StepText.sCode_error[9].ErrorCode := 112;
   // StepText.sCode_error[10].ErrorCode := 122;
   // StepText.sCode_error[11].ErrorCode := 142;
   // StepText.sCode_error[12].ErrorCode := 0;
   // StepText.sCode_error[0].ErrorText := 'Init Step';
   // StepText.sCode_error[1].ErrorText := 'Shuttle EXT Sequence';
   // StepText.sCode_error[2].ErrorText := 'EXT Load/Unload Sequence';
   // StepText.sCode_error[3].ErrorText := 'Part Control In Sequence';
   // StepText.sCode_error[4].ErrorText := 'BW Load Sequence';
   // StepText.sCode_error[5].ErrorText := 'BW Control  Sequence';
   // StepText.sCode_error[6].ErrorText := 'Shuttle INT Sequence';
   // StepText.sCode_error[7].ErrorText := 'INT Load/Unload Sequence';
   // StepText.sCode_error[8].ErrorText := 'Shuttle EXT Sequence';
   // StepText.sCode_error[9].ErrorText := 'BW Unload Sequence';
   // StepText.sCode_error[10].ErrorText := 'Part Control Out Sequence';
   // StepText.sCode_error[11].ErrorText := 'Shuttle INT Sequence';
   // StepText.sCode_error[12].ErrorText := '';
BEGIN
   REGION Description header 
       //==================================================================================
       // POSALUX Swiss SA / (C) Copyright 2025
       //----------------------------------------------------------------------------------
       // Title: FB_Washing
       // Comment/Function: 
       // Author: Fabien WALDT
       // Engineering: TIA Portal v17
       //----------------------------------------------------------------------------------
       // Change log table:
       // Version  | Date     | Expert in charge | Changes applied
       // ---------|----------|------------------|-----------------------------------------
       // 00.00.01 | 20250527 | WFA              | First released version
       // =================================================================================
   END_REGION

   REGION Define condition to start
       IF #iStartSeqCond THEN
           #sInterface.SequenceReleased := TRUE;
       ELSE
           // Standard sequencer controls
           #sInterface.SequenceReleased := FALSE;
           #sCurrent_Step_NB := #S00_INIT_STEP;
           #sInterface.SequenceRun := FALSE;
           #sInterface.JobDone := FALSE;
           #sCheck_Step_Condition := FALSE;

           // Dedicated sequencer controls
           #ioShuttleIntSeq.StartRequest := FALSE;
           #ioShuttleExtSeq.StartRequest := FALSE;
           #ioControlInSeq.StartRequest := FALSE;
           #ioControlOutSeq.StartRequest := FALSE;
           #ioIntLoadUnloadSeq.StartRequest := FALSE;
           #ioExtLoadUnloadSeq.StartRequest := FALSE;
           #ioBWLoadUnloadSeq.StartRequest := FALSE;
           #ioBWControlSeq.StartRequest := FALSE;
           #ioActBwControlInSeq.StartRequest := FALSE;
           #ioActPartControlInSeq.StartRequest := FALSE;
           #ioActPartControlOutSeq.StartRequest := FALSE;
           #sGripperAxisRequest := FALSE;
           #sGripperAxisRelease := TRUE;
           #oNoExtLoad := FALSE;
           #oBwLoadReq := FALSE;
           #oBwUnloadReq := FALSE;
           #ioIntLoadUnloadOP_Seq.StartRequest := FALSE;
           // Add specifics controls 
       END_IF;

       // Reset interface error 
       IF #sInterface.Reset THEN
           #sInterface.Error := FALSE;
       END_IF;

       // One step forward
       #sRTOneStepForward.CLK := #sOneStepForward;
       #sRTOneStepForward();
       #sStepForward := (NOT #sOneStepMode OR (#sOneStepMode AND #sRTOneStepForward.Q)) AND NOT #iStepPause;
       #sOneStepForward := FALSE;
   END_REGION

   REGION Sequence Function
       CASE #sCurrent_Step_NB OF
           #S00_INIT_STEP:
               REGION S00 INIT
                   #sCheck_Step_Condition := TRUE;
               END_REGION
           #S10_SHUTTLE_EXT_SEQ_REQUEST:
               REGION S10_SHUTTLE_EXT_SEQ_REQUEST
                   #ioShuttleExtSeq.StartRequest := TRUE;
                   #sCheck_Step_Condition := TRUE;
               END_REGION
           #S12_SHUTTLE_EXT_SEQ_IN_PROGRESS:
               REGION S12_SHUTTLE_EXT_SEQ_IN_PROGRESS
                   #sCheck_Step_Condition := TRUE;
               END_REGION
           #S14_SHUTTLE_EXT_SEQ_ACQUIT:
               REGION S14_SHUTTLE_EXT_SEQ_ACQUIT
                   #ioShuttleExtSeq.StartRequest := FALSE;
                   #sCheck_Step_Condition := TRUE;
               END_REGION
           #S19_SHUTTLE_EXT_SEQ_ERROR:
               REGION S19_SHUTTLE_EXT_SEQ_ERROR
                   #sCheck_Step_Condition := TRUE;
               END_REGION

           #S20_EXT_LOAD_UNLOAD_SEQ_REQUEST:
               REGION S20_EXT_LOAD_UNLOAD_SEQ_REQUEST
                   #ioExtLoadUnloadSeq.StartRequest := TRUE;
                   #sCheck_Step_Condition := TRUE;
               END_REGION
           #S22_EXT_LOAD_UNLOAD_SEQ_IN_PROGRESS:
               REGION S22_EXT_LOAD_UNLOAD_SEQ_IN_PROGRESS
                   #sCheck_Step_Condition := TRUE;
               END_REGION
           #S24_EXT_LOAD_UNLOAD_SEQ_ACQUIT:
               REGION S24_EXT_LOAD_UNLOAD_SEQ_ACQUIT
                   #ioExtLoadUnloadSeq.StartRequest := FALSE;
                   #sCheck_Step_Condition := TRUE;
               END_REGION
           #S29_EXT_LOAD_UNLOAD_SEQ_ERROR:
               REGION S29_EXT_LOAD_UNLOAD_SEQ_ERROR
                   #sCheck_Step_Condition := TRUE;
               END_REGION

           #S30_PARTS_CTRL_IN_SEQ_REQUEST:
               REGION S30_PARTS_CTRL_IN_SEQ_REQUEST
                   #ioControlInSeq.StartRequest := TRUE;
                   #sCheck_Step_Condition := TRUE;
               END_REGION
           #S32_PARTS_CTRL_IN_SEQ_IN_PROGRESS:
               REGION S32_PARTS_CTRL_IN_SEQ_IN_PROGRESS
                   #sCheck_Step_Condition := TRUE;
               END_REGION
           #S34_PARTS_CTRL_IN_SEQ_ACQUIT:
               REGION S34_PARTS_CTRL_IN_SEQ_ACQUIT
                   #ioControlInSeq.StartRequest := FALSE;
                   #sCheck_Step_Condition := TRUE;
               END_REGION
           #S39_PARTS_CTRL_IN_SEQ_ERROR:
               REGION S39_PARTS_CTRL_IN_SEQ_ERROR
                   #sCheck_Step_Condition := TRUE;
               END_REGION

           #S40_BW_LOAD_UNLOAD_SEQ_REQUEST:
               REGION S40_BW_LOAD_UNLOAD_SEQ_REQUEST
                   #ioBWLoadUnloadSeq.StartRequest := TRUE;
                   IF #iShuttleUndrilledPart AND NOT #iShuttleUndrilledBw THEN
                       #oBwLoadReq := TRUE;
                   END_IF;
                   #sCheck_Step_Condition := TRUE;
               END_REGION
           #S42_BW_LOAD_UNLOAD_SEQ_IN_PROGRESS:
               REGION S42_BW_LOAD_UNLOAD_SEQ_IN_PROGRESS
                   IF #iShuttleUndrilledPart AND NOT #iShuttleUndrilledBw THEN
                       #oBwLoadReq := TRUE;
                   END_IF;
                   #sCheck_Step_Condition := TRUE;
               END_REGION
           #S44_BW_LOAD_UNLOAD_SEQ_ACQUIT:
               REGION S44_BW_LOAD_UNLOAD_SEQ_ACQUIT
                   #ioBWLoadUnloadSeq.StartRequest := FALSE;
                   #oBwLoadReq := FALSE;
                   #sCheck_Step_Condition := TRUE;
               END_REGION
           #S49_BW_LOAD_UNLOAD_SEQ_ERROR:
               REGION S49_BW_LOAD_UNLOAD_SEQ_ERROR
                   #oBwLoadReq := FALSE;
                   #sCheck_Step_Condition := TRUE;
               END_REGION

           #S50_BW_CTRL_UNLOAD_SEQ_REQUEST:
               REGION S50_BW_CTRL_UNLOAD_SEQ_REQUEST
                   #ioBWControlSeq.StartRequest := TRUE;
                   #sCheck_Step_Condition := TRUE;
               END_REGION
           #S52_BW_CTRL_UNLOAD_SEQ_IN_PROGRESS:
               REGION S52_BW_CTRL_UNLOAD_SEQ_IN_PROGRESS
                   #sCheck_Step_Condition := TRUE;
               END_REGION
           #S54_BW_CTRL_UNLOAD_SEQ_ACQUIT:
               REGION S54_BW_CTRL_UNLOAD_SEQ_ACQUIT
                   #ioBWControlSeq.StartRequest := FALSE;
                   #sCheck_Step_Condition := TRUE;
               END_REGION
           #S59_BW_CTRL_UNLOAD_SEQ_ERROR:
               REGION S59_BW_CTRL_UNLOAD_SEQ_ERROR
                   #sCheck_Step_Condition := TRUE;
               END_REGION

           #S60_SHUTTLE_INT_SEQ_REQUEST:
               REGION S60_SHUTTLE_INT_SEQ_REQUEST
                   #ioShuttleIntSeq.StartRequest := TRUE;
                   #sCheck_Step_Condition := TRUE;
               END_REGION
           #S62_SHUTTLE_INT_SEQ_IN_PROGRESS:
               REGION S62_SHUTTLE_INT_SEQ_IN_PROGRESS
                   #sCheck_Step_Condition := TRUE;
               END_REGION
           #S64_SHUTTLE_INT_SEQ_ACQUIT:
               REGION S64_SHUTTLE_INT_SEQ_ACQUIT
                   #ioShuttleIntSeq.StartRequest := FALSE;
                   #sCheck_Step_Condition := TRUE;
               END_REGION
           #S69_SHUTTLE_INT_SEQ_ERROR:
               REGION S69_SHUTTLE_INT_SEQ_ERROR
                   #sCheck_Step_Condition := TRUE;
               END_REGION

           #S70_TRANSFER_V_AND_W_AXIS_TO_PLC:
               REGION S70_TRANSFER_V_AND_W_AXIS_TO_PLC
                   IF #iGripperOK THEN
                       #sGripperAxisRequest := TRUE;
                       #sGripperAxisRelease := FALSE;
                       #sCheck_Step_Condition := TRUE;
                   END_IF;
                   END_REGION

           #S80_INT_LOAD_UNLOAD_SEQ_REQUEST:
               REGION S80_INT_LOAD_UNLOAD_SEQ_REQUEST
                   #ioIntLoadUnloadSeq.StartRequest := TRUE;
                   #sCheck_Step_Condition := TRUE;
               END_REGION
           #S82_INT_LOAD_UNLOAD_SEQ_IN_PROGRESS:
               REGION S82_INT_LOAD_UNLOAD_SEQ_IN_PROGRESS
                   #sCheck_Step_Condition := TRUE;
               END_REGION
           #S84_INT_LOAD_UNLOAD_SEQ_ACQUIT:
               REGION S84_INT_LOAD_UNLOAD_SEQ_ACQUIT
                   #ioIntLoadUnloadSeq.StartRequest := FALSE;
                   #sCheck_Step_Condition := TRUE;
               END_REGION
           #S89_INT_LOAD_UNLOAD_SEQ_ERROR:
               REGION S89_INT_LOAD_UNLOAD_SEQ_ERROR
                   #sCheck_Step_Condition := TRUE;
               END_REGION

           #S90_TRANSFER_V_AND_W_AXIS_TO_NC:
               REGION S90_TRANSFER_V_AND_W_AXIS_TO_NC
                   #sGripperAxisRequest := FALSE;
                   #sGripperAxisRelease := TRUE;
                   #sCheck_Step_Condition := TRUE;
               END_REGION

           #S100_SHUTTLE_EXT_SEQ_REQUEST:
               REGION S100_SHUTTLE_EXT_SEQ_REQUEST
                   #ioShuttleExtSeq.StartRequest := TRUE;
                   #sCheck_Step_Condition := TRUE;
               END_REGION
           #S102_SHUTTLE_EXT_SEQ_IN_PROGRESS:
               REGION S102_SHUTTLE_EXT_SEQ_IN_PROGRESS
                   #sCheck_Step_Condition := TRUE;
               END_REGION
           #S104_SHUTTLE_EXT_SEQ_ACQUIT:
               REGION S104_SHUTTLE_EXT_SEQ_ACQUIT
                   #ioShuttleExtSeq.StartRequest := FALSE;
                   #sCheck_Step_Condition := TRUE;
               END_REGION
           #S109_SHUTTLE_EXT_SEQ_ERROR:
               REGION S109_SHUTTLE_EXT_SEQ_ERROR
                   #sCheck_Step_Condition := TRUE;
               END_REGION

           #S110_BW_LOAD_UNLOAD_SEQ_REQUEST:
               REGION S110_BW_LOAD_UNLOAD_SEQ_REQUEST
                   #ioBWLoadUnloadSeq.StartRequest := TRUE;
                   IF #iShuttleDrilledBw THEN
                       #oBwUnloadReq := TRUE;
                   END_IF;
                   #sCheck_Step_Condition := TRUE;
               END_REGION
           #S112_BW_LOAD_UNLOAD_SEQ_IN_PROGRESS:
               REGION S112_BW_LOAD_UNLOAD_SEQ_IN_PROGRESS
                   IF #iShuttleDrilledBw THEN
                       #oBwUnloadReq := TRUE;
                   END_IF;
                   #sCheck_Step_Condition := TRUE;
               END_REGION
           #S114_BW_LOAD_UNLOAD_SEQ_ACQUIT:
               REGION S114_BW_LOAD_UNLOAD_SEQ_ACQUIT
                   #ioBWLoadUnloadSeq.StartRequest := FALSE;
                   #oBwUnloadReq := FALSE;
                   #sCheck_Step_Condition := TRUE;
               END_REGION
           #S119_BW_LOAD_UNLOAD_SEQ_ERROR:
               REGION S119_BW_LOAD_UNLOAD_SEQ_ERROR
                   #oBwUnloadReq := FALSE;
                   #sCheck_Step_Condition := TRUE;
               END_REGION

           #S120_PARTS_CTRL_OUT_SEQ_REQUEST:
               REGION S120_PARTS_CTRL_OUT_SEQ_REQUEST
                   #ioControlOutSeq.StartRequest := TRUE;
                   #sCheck_Step_Condition := TRUE;
               END_REGION
           #S122_PARTS_CTRL_OUT_SEQ_IN_PROGRESS:
               REGION S122_PARTS_CTRL_OUT_SEQ_IN_PROGRESS
                   #sCheck_Step_Condition := TRUE;
               END_REGION
           #S124_PARTS_CTRL_OUT_SEQ_ACQUIT:
               REGION S124_PARTS_CTRL_OUT_SEQ_ACQUIT
                   #ioControlOutSeq.StartRequest := FALSE;
                   #sCheck_Step_Condition := TRUE;
               END_REGION
           #S129_PARTS_CTRL_OUT_SEQ_ERROR:
               REGION S129_PARTS_CTRL_OUT_SEQ_ERROR
                   #sCheck_Step_Condition := TRUE;
               END_REGION

           #S130_CHECK_CYCLE_STOP:
               REGION S130_CHECK_CYCLE_STOP
                   #sCheck_Step_Condition := TRUE;
               END_REGION

           #S140_EXT_LOAD_UNLOAD_SEQ_REQUEST:
               REGION S140_EXT_LOAD_UNLOAD_SEQ_REQUEST
                   #ioExtLoadUnloadSeq.StartRequest := TRUE;
                   #oNoExtLoad := TRUE;
                   #sCheck_Step_Condition := TRUE;
               END_REGION
           #S142_EXT_LOAD_UNLOAD_SEQ_IN_PROGRESS:
               REGION S142_EXT_LOAD_UNLOAD_SEQ_IN_PROGRESS
                   #sCheck_Step_Condition := TRUE;
               END_REGION
           #S144_EXT_LOAD_UNLOAD_SEQ_ACQUIT:
               REGION S144_EXT_LOAD_UNLOAD_SEQ_ACQUIT
                   #ioExtLoadUnloadSeq.StartRequest := FALSE;
                   #oNoExtLoad := FALSE;
                   #sCheck_Step_Condition := TRUE;
               END_REGION
           #S149_EXT_LOAD_UNLOAD_SEQ_ERROR:
               REGION S149_EXT_LOAD_UNLOAD_SEQ_ERROR
                   #oNoExtLoad := FALSE;
                   #sCheck_Step_Condition := TRUE;
               END_REGION

           #S200_BLOWING_SEQ_REQUEST:
               REGION S200_BLOWING_SEQ_REQUEST
                   #ioBlowingSeq.StartRequest := TRUE;
                   #sCheck_Step_Condition := TRUE;
               END_REGION
           #S202_BLOWING_SEQ_IN_PROGRESS:
               REGION S202_BLOWING_SEQ_IN_PROGRESS
                   #sCheck_Step_Condition := TRUE;
               END_REGION
           #S204_BLOWING_SEQ_ACQUIT:
               REGION S204_BLOWING_SEQ_ACQUIT
                   #ioBlowingSeq.StartRequest := FALSE;
                   #sCheck_Step_Condition := TRUE;
               END_REGION
           #S209_BLOWING_SEQ_ERROR:
               REGION S209_BLOWING_SEQ_ERROR
                   #sCheck_Step_Condition := TRUE;
               END_REGION

           #S210_INT_LOAD_UNLOAD_OP_SEQ_REQUEST:
               REGION S210_INT_LOAD_UNLOAD_OP_SEQ_REQUEST
                   #ioIntLoadUnloadOP_Seq.StartRequest := TRUE;
                   #sCheck_Step_Condition := TRUE;
               END_REGION
           #S212_INT_LOAD_UNLOAD_OP_SEQ_IN_PROGRESS:
               REGION S212_INT_LOAD_UNLOAD_OP_SEQ_IN_PROGRESS
                   #sCheck_Step_Condition := TRUE;
               END_REGION
           #S214_INT_LOAD_UNLOAD_OP_SEQ_ACQUIT:
               REGION S214_INT_LOAD_UNLOAD_OP_SEQ_ACQUIT
                   #ioIntLoadUnloadOP_Seq.StartRequest := FALSE;
                   #sCheck_Step_Condition := TRUE;
               END_REGION
           #S219_INT_LOAD_UNLOAD_OP_SEQ_ERROR:
               REGION S219_INT_LOAD_UNLOAD_OP_SEQ_ERROR
                   #sCheck_Step_Condition := TRUE;
               END_REGION

           #S300_ACT_PART_CTRL_IN_SEQ_REQUEST:
               REGION S300_ACT_PART_CTRL_IN_SEQ_REQUEST
                   #ioActPartControlInSeq.StartRequest := TRUE;
                   #sCheck_Step_Condition := TRUE;
               END_REGION
           #S302_ACT_PART_CTRL_IN_SEQ_IN_PROGRESS:
               REGION S302_ACT_PART_CTRL_IN_SEQ_IN_PROGRESS
                   #sCheck_Step_Condition := TRUE;
               END_REGION
           #S304_ACT_PART_CTRL_IN_SEQ_ACQUIT:
               REGION S304_ACT_PART_CTRL_IN_SEQ_ACQUIT
                   #ioActPartControlInSeq.StartRequest := FALSE;
                   #sCheck_Step_Condition := TRUE;
               END_REGION
           #S309_ACT_PART_CTRL_IN_SEQ_ERROR:
               REGION S309_ACT_PART_CTRL_IN_SEQ_ERROR
                   #sCheck_Step_Condition := TRUE;
               END_REGION

           #S310_ACT_PART_CTRL_OUT_SEQ_REQUEST:
               REGION S310_ACT_PART_CTRL_OUT_SEQ_REQUEST
                   #ioActPartControlOutSeq.StartRequest := TRUE;
                   #sCheck_Step_Condition := TRUE;
               END_REGION
           #S312_ACT_PART_CTRL_OUT_SEQ_IN_PROGRESS:
               REGION S312_ACT_PART_CTRL_OUT_SEQ_IN_PROGRESS
                   #sCheck_Step_Condition := TRUE;
               END_REGION
           #S314_ACT_PART_CTRL_OUT_SEQ_ACQUIT:
               REGION S314_ACT_PART_CTRL_OUT_SEQ_ACQUIT
                   #ioActPartControlOutSeq.StartRequest := FALSE;
                   #sCheck_Step_Condition := TRUE;
               END_REGION
           #S319_ACT_PART_CTRL_OUT_SEQ_ERROR:
               REGION S319_ACT_PART_CTRL_OUT_SEQ_ERROR
                   #sCheck_Step_Condition := TRUE;
               END_REGION

           #S320_ACT_BW_CTRL_IN_SEQ_REQUEST:
               REGION S320_ACT_BW_CTRL_IN_SEQ_REQUEST
                   #ioActBwControlInSeq.StartRequest := TRUE;
                   #sCheck_Step_Condition := TRUE;
               END_REGION
           #S322_ACT_BW_CTRL_IN_SEQ_IN_PROGRESS:
               REGION S322_ACT_BW_CTRL_IN_SEQ_IN_PROGRESS
                   #sCheck_Step_Condition := TRUE;
               END_REGION
           #S324_ACT_BW_CTRL_IN_SEQ_ACQUIT:
               REGION S324_ACT_BW_CTRL_IN_SEQ_ACQUIT
                   #ioActBwControlInSeq.StartRequest := FALSE;
                   #sCheck_Step_Condition := TRUE;
               END_REGION
           #S329_ACT_BW_CTRL_IN_SEQ_ERROR:
               REGION S329_ACT_BW_CTRL_IN_SEQ_ERROR
                   #sCheck_Step_Condition := TRUE;
               END_REGION

           #S999_ERROR:
               REGION S999_ERROR
                   #sCheck_Step_Condition := TRUE;
               END_REGION
           ELSE:
               #sInterface.Error := TRUE;
       END_CASE;
   END_REGION

   REGION Sequence Next Step Condition
       IF #sCheck_Step_Condition THEN
           CASE #sCurrent_Step_NB OF
               #S00_INIT_STEP:
                   REGION S00 INIT
                       IF #sInterface.SequenceReleased AND #iJobReq AND NOT #iShuttleUndrilledPart AND NOT #iShuttleDrilledPart AND (#iShuttleEXT) THEN
                           #sCurrent_Step_NB := #S10_SHUTTLE_EXT_SEQ_REQUEST;
                           #sInterface.SequenceRun := TRUE;
                           #sCheck_Step_Condition := FALSE;
                       ELSIF #sInterface.SequenceReleased AND #iJobReq AND #iShuttleUndrilledPart AND NOT #iShuttleUndrilledBw AND NOT #iShuttleDrilledPart THEN
                           #sCurrent_Step_NB := #S30_PARTS_CTRL_IN_SEQ_REQUEST;
                           #sInterface.SequenceRun := TRUE;
                           #sCheck_Step_Condition := FALSE;
                       ELSIF #sInterface.SequenceReleased AND #iJobReq AND #iShuttleEXT AND #iShuttleUndrilledPart AND #iShuttleUndrilledBw AND NOT #iShuttleDrilledPart THEN
                           #sCurrent_Step_NB := #S50_BW_CTRL_UNLOAD_SEQ_REQUEST;
                           #sInterface.SequenceRun := TRUE;
                           #sCheck_Step_Condition := FALSE;
                       ELSIF #sInterface.SequenceReleased AND #iJobReq AND (#iShuttleSAS OR #iShuttleINT) AND #iShuttleUndrilledPart AND #iShuttleUndrilledBw AND NOT #iShuttleDrilledPart THEN
                           #sCurrent_Step_NB := #S60_SHUTTLE_INT_SEQ_REQUEST;
                           #sInterface.SequenceRun := TRUE;
                           #sCheck_Step_Condition := FALSE;
                       ELSIF #sInterface.SequenceReleased AND #iJobReq AND (((#iShuttleSAS OR #iShuttleINT) AND NOT #iShuttleUndrilledPart AND #iShuttleDrilledPart AND #iShuttleDrilledBw)
                           OR #sInterface.SequenceReleased AND #iJobReq AND NOT #iShuttleUndrilledPart AND NOT #iShuttleDrilledPart AND (#iShuttleSAS OR #iShuttleINT)
                           OR ((#iShuttleSAS OR #iShuttleINT) AND NOT #iShuttleUndrilledPart AND #iShuttleDrilledPart AND NOT #iShuttleDrilledBw)) THEN
                           #sCurrent_Step_NB := #S100_SHUTTLE_EXT_SEQ_REQUEST;
                           #sInterface.SequenceRun := TRUE;
                           #sCheck_Step_Condition := FALSE;
                       ELSIF #sInterface.SequenceReleased AND #iJobReq AND #iShuttleEXT AND NOT #iShuttleUndrilledPart AND #iShuttleDrilledPart AND #iShuttleDrilledBw THEN
                           #sCurrent_Step_NB := #S110_BW_LOAD_UNLOAD_SEQ_REQUEST;
                           #sInterface.SequenceRun := TRUE;
                           #sCheck_Step_Condition := FALSE;
                       ELSIF #sInterface.SequenceReleased AND #iJobReq AND #iShuttleEXT AND NOT #iShuttleUndrilledPart AND #iShuttleDrilledPart AND NOT #iShuttleDrilledBw THEN
                           #sCurrent_Step_NB := #S120_PARTS_CTRL_OUT_SEQ_REQUEST;
                           #sInterface.SequenceRun := TRUE;
                           #sCheck_Step_Condition := FALSE;
                       ELSE
                           #sInterface.SequenceRun := FALSE;
                       END_IF;
                   END_REGION

               #S10_SHUTTLE_EXT_SEQ_REQUEST:
                   REGION S10_SHUTTLE_EXT_SEQ_REQUEST
                       IF #sInterface.SequenceReleased AND #ioShuttleExtSeq.SequenceRun THEN
                           #sCurrent_Step_NB := #S12_SHUTTLE_EXT_SEQ_IN_PROGRESS;
                           #sCheck_Step_Condition := FALSE;
                       ELSIF #sInterface.SequenceReleased AND #ioShuttleExtSeq.Error THEN
                           #sCurrent_Step_NB := #S19_SHUTTLE_EXT_SEQ_ERROR;
                           #sCheck_Step_Condition := FALSE;
                       END_IF;
                   END_REGION
               #S12_SHUTTLE_EXT_SEQ_IN_PROGRESS:
                   REGION S12_SHUTTLE_EXT_SEQ_IN_PROGRESS
                       IF #sInterface.SequenceReleased AND #ioShuttleExtSeq.JobDone THEN
                           #sCurrent_Step_NB := #S14_SHUTTLE_EXT_SEQ_ACQUIT;
                           #sCheck_Step_Condition := FALSE;
                       ELSIF #sInterface.SequenceReleased AND #ioShuttleExtSeq.Error THEN
                           #sCurrent_Step_NB := #S19_SHUTTLE_EXT_SEQ_ERROR;
                           #sCheck_Step_Condition := FALSE;
                       END_IF;
                   END_REGION
               #S14_SHUTTLE_EXT_SEQ_ACQUIT:
                   REGION S14_SHUTTLE_EXT_SEQ_ACQUIT
                       IF #sInterface.SequenceReleased AND "AlwaysTRUE" THEN
                           #sCurrent_Step_NB := #S20_EXT_LOAD_UNLOAD_SEQ_REQUEST;
                           #sCheck_Step_Condition := FALSE;
                       END_IF;
                   END_REGION
               #S19_SHUTTLE_EXT_SEQ_ERROR:
                   REGION S19_SHUTTLE_EXT_SEQ_ERROR
                       IF #sInterface.SequenceReleased AND "AlwaysTRUE" THEN
                           #sCurrent_Step_NB := #S999_ERROR;
                           #sCheck_Step_Condition := FALSE;
                       END_IF;
                   END_REGION

               #S20_EXT_LOAD_UNLOAD_SEQ_REQUEST:
                   REGION S20_EXT_LOAD_UNLOAD_SEQ_REQUEST
                       IF #sInterface.SequenceReleased AND #ioExtLoadUnloadSeq.SequenceRun THEN
                           #sCurrent_Step_NB := #S22_EXT_LOAD_UNLOAD_SEQ_IN_PROGRESS;
                           #sCheck_Step_Condition := FALSE;
                       ELSIF #sInterface.SequenceReleased AND #ioExtLoadUnloadSeq.Error THEN
                           #sCurrent_Step_NB := #S29_EXT_LOAD_UNLOAD_SEQ_ERROR;
                           #sCheck_Step_Condition := FALSE;
                       END_IF;
                   END_REGION
               #S22_EXT_LOAD_UNLOAD_SEQ_IN_PROGRESS:
                   REGION S22_EXT_LOAD_UNLOAD_SEQ_IN_PROGRESS
                       IF #sInterface.SequenceReleased AND #ioExtLoadUnloadSeq.JobDone THEN
                           #sCurrent_Step_NB := #S24_EXT_LOAD_UNLOAD_SEQ_ACQUIT;
                           #sCheck_Step_Condition := FALSE;
                       ELSIF #sInterface.SequenceReleased AND #ioExtLoadUnloadSeq.Error THEN
                           #sCurrent_Step_NB := #S29_EXT_LOAD_UNLOAD_SEQ_ERROR;
                           #sCheck_Step_Condition := FALSE;
                       END_IF;
                   END_REGION
               #S24_EXT_LOAD_UNLOAD_SEQ_ACQUIT:
                   REGION S24_EXT_LOAD_UNLOAD_SEQ_ACQUIT
                       IF #sInterface.SequenceReleased AND "AlwaysTRUE" THEN
                           #sCurrent_Step_NB := #S30_PARTS_CTRL_IN_SEQ_REQUEST;
                           #sCheck_Step_Condition := FALSE;
                       END_IF;
                   END_REGION
               #S29_EXT_LOAD_UNLOAD_SEQ_ERROR:
                   REGION S29_EXT_LOAD_UNLOAD_SEQ_ERROR
                       IF #sInterface.SequenceReleased AND "AlwaysTRUE" THEN
                           #sCurrent_Step_NB := #S999_ERROR;
                           #sCheck_Step_Condition := FALSE;
                       END_IF;
                   END_REGION

               #S30_PARTS_CTRL_IN_SEQ_REQUEST:
                   REGION S30_PARTS_CTRL_IN_SEQ_REQUEST
                       IF #sInterface.SequenceReleased AND #ioControlInSeq.SequenceRun THEN
                           #sCurrent_Step_NB := #S32_PARTS_CTRL_IN_SEQ_IN_PROGRESS;
                           #sCheck_Step_Condition := FALSE;
                       ELSIF #sInterface.SequenceReleased AND #ioControlInSeq.Error THEN
                           #sCurrent_Step_NB := #S39_PARTS_CTRL_IN_SEQ_ERROR;
                           #sCheck_Step_Condition := FALSE;
                       END_IF;
                   END_REGION
               #S32_PARTS_CTRL_IN_SEQ_IN_PROGRESS:
                   REGION S32_PARTS_CTRL_IN_SEQ_IN_PROGRESS
                       IF #sInterface.SequenceReleased AND #ioControlInSeq.JobDone THEN
                           #sCurrent_Step_NB := #S34_PARTS_CTRL_IN_SEQ_ACQUIT;
                           #sCheck_Step_Condition := FALSE;
                       ELSIF #sInterface.SequenceReleased AND #ioControlInSeq.Error THEN
                           #sCurrent_Step_NB := #S39_PARTS_CTRL_IN_SEQ_ERROR;
                           #sCheck_Step_Condition := FALSE;
                       END_IF;
                   END_REGION
               #S34_PARTS_CTRL_IN_SEQ_ACQUIT:
                   REGION S34_PARTS_CTRL_IN_SEQ_ACQUIT
                       IF #sInterface.SequenceReleased AND #iPartCtrlInOK AND NOT #iPartCtrlInNOK THEN
                           #sCurrent_Step_NB := #S40_BW_LOAD_UNLOAD_SEQ_REQUEST;
                           #sCheck_Step_Condition := FALSE;
                       ELSIF #sInterface.SequenceReleased AND NOT #iPartCtrlInOK AND #iPartCtrlInNOK THEN
                           #sCurrent_Step_NB := #S300_ACT_PART_CTRL_IN_SEQ_REQUEST;
                           #sCheck_Step_Condition := FALSE;
                       END_IF;
                   END_REGION
               #S39_PARTS_CTRL_IN_SEQ_ERROR:
                   REGION S39_PARTS_CTRL_IN_SEQ_ERROR
                       IF #sInterface.SequenceReleased AND "AlwaysTRUE" THEN
                           #sCurrent_Step_NB := #S999_ERROR;
                           #sCheck_Step_Condition := FALSE;
                       END_IF;
                   END_REGION

               #S40_BW_LOAD_UNLOAD_SEQ_REQUEST:
                   REGION S40_BW_LOAD_UNLOAD_SEQ_REQUEST
                       IF #sInterface.SequenceReleased AND #ioBWLoadUnloadSeq.SequenceRun THEN
                           #sCurrent_Step_NB := #S42_BW_LOAD_UNLOAD_SEQ_IN_PROGRESS;
                           #sCheck_Step_Condition := FALSE;
                       ELSIF #sInterface.SequenceReleased AND #ioBWLoadUnloadSeq.Error THEN
                           #sCurrent_Step_NB := #S49_BW_LOAD_UNLOAD_SEQ_ERROR;
                           #sCheck_Step_Condition := FALSE;
                       END_IF;
                   END_REGION
               #S42_BW_LOAD_UNLOAD_SEQ_IN_PROGRESS:
                   REGION S42_BW_LOAD_UNLOAD_SEQ_IN_PROGRESS
                       IF #sInterface.SequenceReleased AND #ioBWLoadUnloadSeq.JobDone THEN
                           #sCurrent_Step_NB := #S44_BW_LOAD_UNLOAD_SEQ_ACQUIT;
                           #sCheck_Step_Condition := FALSE;
                       ELSIF #sInterface.SequenceReleased AND #ioBWLoadUnloadSeq.Error THEN
                           #sCurrent_Step_NB := #S49_BW_LOAD_UNLOAD_SEQ_ERROR;
                           #sCheck_Step_Condition := FALSE;
                       END_IF;
                   END_REGION
               #S44_BW_LOAD_UNLOAD_SEQ_ACQUIT:
                   REGION S44_BW_LOAD_UNLOAD_SEQ_ACQUIT
                       IF #sInterface.SequenceReleased AND "AlwaysTRUE" THEN
                           #sCurrent_Step_NB := #S50_BW_CTRL_UNLOAD_SEQ_REQUEST;
                           #sCheck_Step_Condition := FALSE;
                       END_IF;
                   END_REGION
               #S49_BW_LOAD_UNLOAD_SEQ_ERROR:
                   REGION S49_BW_LOAD_UNLOAD_SEQ_ERROR
                       IF #sInterface.SequenceReleased AND "AlwaysTRUE" THEN
                           #sCurrent_Step_NB := #S999_ERROR;
                           #sCheck_Step_Condition := FALSE;
                       END_IF;
                   END_REGION

               #S50_BW_CTRL_UNLOAD_SEQ_REQUEST:
                   REGION S50_BW_CTRL_UNLOAD_SEQ_REQUEST
                       IF #sInterface.SequenceReleased AND #ioBWControlSeq.SequenceRun THEN
                           #sCurrent_Step_NB := #S52_BW_CTRL_UNLOAD_SEQ_IN_PROGRESS;
                           #sCheck_Step_Condition := FALSE;
                       ELSIF #sInterface.SequenceReleased AND #ioBWControlSeq.Error THEN
                           #sCurrent_Step_NB := #S59_BW_CTRL_UNLOAD_SEQ_ERROR;
                           #sCheck_Step_Condition := FALSE;
                       END_IF;
                   END_REGION
               #S52_BW_CTRL_UNLOAD_SEQ_IN_PROGRESS:
                   REGION S52_BW_CTRL_UNLOAD_SEQ_IN_PROGRESS
                       IF #sInterface.SequenceReleased AND #ioBWControlSeq.JobDone THEN
                           #sCurrent_Step_NB := #S54_BW_CTRL_UNLOAD_SEQ_ACQUIT;
                           #sCheck_Step_Condition := FALSE;
                       ELSIF #sInterface.SequenceReleased AND #ioBWControlSeq.Error THEN
                           #sCurrent_Step_NB := #S59_BW_CTRL_UNLOAD_SEQ_ERROR;
                           #sCheck_Step_Condition := FALSE;
                       END_IF;
                   END_REGION
               #S54_BW_CTRL_UNLOAD_SEQ_ACQUIT:
                   REGION S54_BW_CTRL_UNLOAD_SEQ_ACQUIT
                       IF #sInterface.SequenceReleased AND #iBwCtrlInOK AND NOT #iBwCtrlInNOK THEN
                           #sCurrent_Step_NB := #S60_SHUTTLE_INT_SEQ_REQUEST;
                           #sCheck_Step_Condition := FALSE;
                       ELSIF #sInterface.SequenceReleased AND NOT #iBwCtrlInOK AND #iBwCtrlInNOK THEN
                           #sCurrent_Step_NB := #S320_ACT_BW_CTRL_IN_SEQ_REQUEST;
                           #sCheck_Step_Condition := FALSE;
                       END_IF;
                   END_REGION
               #S59_BW_CTRL_UNLOAD_SEQ_ERROR:
                   REGION S59_BW_CTRL_UNLOAD_SEQ_ERROR
                       IF #sInterface.SequenceReleased AND "AlwaysTRUE" THEN
                           #sCurrent_Step_NB := #S999_ERROR;
                           #sCheck_Step_Condition := FALSE;
                       END_IF;
                   END_REGION

               #S60_SHUTTLE_INT_SEQ_REQUEST:
                   REGION S60_SHUTTLE_INT_SEQ_REQUEST
                       IF #sInterface.SequenceReleased AND #ioShuttleIntSeq.SequenceRun THEN
                           #sCurrent_Step_NB := #S62_SHUTTLE_INT_SEQ_IN_PROGRESS;
                           #sCheck_Step_Condition := FALSE;
                       ELSIF #sInterface.SequenceReleased AND #ioShuttleIntSeq.Error THEN
                           #sCurrent_Step_NB := #S69_SHUTTLE_INT_SEQ_ERROR;
                           #sCheck_Step_Condition := FALSE;
                       END_IF;
                   END_REGION
               #S62_SHUTTLE_INT_SEQ_IN_PROGRESS:
                   REGION S62_SHUTTLE_INT_SEQ_IN_PROGRESS
                       IF #sInterface.SequenceReleased AND #ioShuttleIntSeq.JobDone THEN
                           #sCurrent_Step_NB := #S64_SHUTTLE_INT_SEQ_ACQUIT;
                           #sCheck_Step_Condition := FALSE;
                       ELSIF #sInterface.SequenceReleased AND #ioShuttleIntSeq.Error THEN
                           #sCurrent_Step_NB := #S69_SHUTTLE_INT_SEQ_ERROR;
                           #sCheck_Step_Condition := FALSE;
                       END_IF;
                   END_REGION
               #S64_SHUTTLE_INT_SEQ_ACQUIT:
                   REGION S64_SHUTTLE_INT_SEQ_ACQUIT
                       IF #sInterface.SequenceReleased AND #iNC_NoNeedAxis THEN
                           #sCurrent_Step_NB := #S70_TRANSFER_V_AND_W_AXIS_TO_PLC;
                           #sCheck_Step_Condition := FALSE;
                       END_IF;
                   END_REGION
               #S69_SHUTTLE_INT_SEQ_ERROR:
                   REGION S69_SHUTTLE_INT_SEQ_ERROR
                       IF #sInterface.SequenceReleased AND "AlwaysTRUE" THEN
                           #sCurrent_Step_NB := #S999_ERROR;
                           #sCheck_Step_Condition := FALSE;
                       END_IF;
                   END_REGION

               #S70_TRANSFER_V_AND_W_AXIS_TO_PLC:
                   REGION S70_TRANSFER_V_AND_W_AXIS_TO_PLC
                       IF #sInterface.SequenceReleased AND #iGripperReserved AND NOT #iGripperReleased AND #iGripperOK THEN
                           #sCurrent_Step_NB := #S200_BLOWING_SEQ_REQUEST;
                           #sCheck_Step_Condition := FALSE;
                       END_IF;
                   END_REGION

               #S80_INT_LOAD_UNLOAD_SEQ_REQUEST:
                   REGION S80_INT_LOAD_UNLOAD_SEQ_REQUEST
                       IF #sInterface.SequenceReleased AND #ioIntLoadUnloadSeq.SequenceRun THEN
                           #sCurrent_Step_NB := #S82_INT_LOAD_UNLOAD_SEQ_IN_PROGRESS;
                           #sCheck_Step_Condition := FALSE;
                       ELSIF #sInterface.SequenceReleased AND #ioIntLoadUnloadSeq.Error THEN
                           #sCurrent_Step_NB := #S89_INT_LOAD_UNLOAD_SEQ_ERROR;
                           #sCheck_Step_Condition := FALSE;
                       END_IF;
                   END_REGION
               #S82_INT_LOAD_UNLOAD_SEQ_IN_PROGRESS:
                   REGION S82_INT_LOAD_UNLOAD_SEQ_IN_PROGRESS
                       IF #sInterface.SequenceReleased AND #ioIntLoadUnloadSeq.JobDone THEN
                           #sCurrent_Step_NB := #S84_INT_LOAD_UNLOAD_SEQ_ACQUIT;
                           #sCheck_Step_Condition := FALSE;
                       ELSIF #sInterface.SequenceReleased AND #ioIntLoadUnloadSeq.Error THEN
                           #sCurrent_Step_NB := #S89_INT_LOAD_UNLOAD_SEQ_ERROR;
                           #sCheck_Step_Condition := FALSE;
                       END_IF;
                   END_REGION
               #S84_INT_LOAD_UNLOAD_SEQ_ACQUIT:
                   REGION S84_INT_LOAD_UNLOAD_SEQ_ACQUIT
                       IF #sInterface.SequenceReleased AND "AlwaysTRUE" THEN
                           #sCurrent_Step_NB := #S90_TRANSFER_V_AND_W_AXIS_TO_NC;
                           #sCheck_Step_Condition := FALSE;
                       END_IF;
                   END_REGION
               #S89_INT_LOAD_UNLOAD_SEQ_ERROR:
                   REGION S89_INT_LOAD_UNLOAD_SEQ_ERROR
                       IF #sInterface.SequenceReleased AND "AlwaysTRUE" THEN
                           #sCurrent_Step_NB := #S999_ERROR;
                           #sCheck_Step_Condition := FALSE;
                       END_IF;
                   END_REGION

               #S90_TRANSFER_V_AND_W_AXIS_TO_NC:
                   REGION S90_TRANSFER_V_AND_W_AXIS_TO_NC
                       IF #sInterface.SequenceReleased AND NOT #iGripperReserved AND #iGripperReleased THEN
                           #sCurrent_Step_NB := #S100_SHUTTLE_EXT_SEQ_REQUEST;
                           #sCheck_Step_Condition := FALSE;
                       END_IF;
                   END_REGION

               #S100_SHUTTLE_EXT_SEQ_REQUEST:
                   REGION S100_SHUTTLE_EXT_SEQ_REQUEST
                       IF #sInterface.SequenceReleased AND #ioShuttleExtSeq.SequenceRun THEN
                           #sCurrent_Step_NB := #S102_SHUTTLE_EXT_SEQ_IN_PROGRESS;
                           #sCheck_Step_Condition := FALSE;
                       ELSIF #sInterface.SequenceReleased AND #ioShuttleExtSeq.Error THEN
                           #sCurrent_Step_NB := #S109_SHUTTLE_EXT_SEQ_ERROR;
                           #sCheck_Step_Condition := FALSE;
                       END_IF;
                   END_REGION
               #S102_SHUTTLE_EXT_SEQ_IN_PROGRESS:
                   REGION S102_SHUTTLE_EXT_SEQ_IN_PROGRESS
                       IF #sInterface.SequenceReleased AND #ioShuttleExtSeq.JobDone THEN
                           #sCurrent_Step_NB := #S104_SHUTTLE_EXT_SEQ_ACQUIT;
                           #sCheck_Step_Condition := FALSE;
                       ELSIF #sInterface.SequenceReleased AND #ioShuttleExtSeq.Error THEN
                           #sCurrent_Step_NB := #S109_SHUTTLE_EXT_SEQ_ERROR;
                           #sCheck_Step_Condition := FALSE;
                       END_IF;
                   END_REGION
               #S104_SHUTTLE_EXT_SEQ_ACQUIT:
                   REGION S104_SHUTTLE_EXT_SEQ_ACQUIT
                       IF #sInterface.SequenceReleased AND "AlwaysTRUE" THEN
                           #sCurrent_Step_NB := #S110_BW_LOAD_UNLOAD_SEQ_REQUEST;
                           #sCheck_Step_Condition := FALSE;
                       END_IF;
                   END_REGION
               #S109_SHUTTLE_EXT_SEQ_ERROR:
                   REGION S109_SHUTTLE_EXT_SEQ_ERROR
                       IF #sInterface.SequenceReleased AND "AlwaysTRUE" THEN
                           #sCurrent_Step_NB := #S999_ERROR;
                           #sCheck_Step_Condition := FALSE;
                       END_IF;
                   END_REGION

               #S110_BW_LOAD_UNLOAD_SEQ_REQUEST:
                   REGION S110_BW_LOAD_UNLOAD_SEQ_REQUEST
                       IF #sInterface.SequenceReleased AND #ioBWLoadUnloadSeq.SequenceRun THEN
                           #sCurrent_Step_NB := #S112_BW_LOAD_UNLOAD_SEQ_IN_PROGRESS;
                           #sCheck_Step_Condition := FALSE;
                       ELSIF #sInterface.SequenceReleased AND #ioBWLoadUnloadSeq.Error THEN
                           #sCurrent_Step_NB := #S119_BW_LOAD_UNLOAD_SEQ_ERROR;
                           #sCheck_Step_Condition := FALSE;
                       END_IF;
                   END_REGION
               #S112_BW_LOAD_UNLOAD_SEQ_IN_PROGRESS:
                   REGION S112_BW_LOAD_UNLOAD_SEQ_IN_PROGRESS
                       IF #sInterface.SequenceReleased AND #ioBWLoadUnloadSeq.JobDone THEN
                           #sCurrent_Step_NB := #S114_BW_LOAD_UNLOAD_SEQ_ACQUIT;
                           #sCheck_Step_Condition := FALSE;
                       ELSIF #sInterface.SequenceReleased AND #ioBWLoadUnloadSeq.Error THEN
                           #sCurrent_Step_NB := #S119_BW_LOAD_UNLOAD_SEQ_ERROR;
                           #sCheck_Step_Condition := FALSE;
                       END_IF;
                   END_REGION
               #S114_BW_LOAD_UNLOAD_SEQ_ACQUIT:
                   REGION S114_BW_LOAD_UNLOAD_SEQ_ACQUIT
                       IF #sInterface.SequenceReleased AND "AlwaysTRUE" THEN
                           #sCurrent_Step_NB := #S120_PARTS_CTRL_OUT_SEQ_REQUEST;
                           #sCheck_Step_Condition := FALSE;
                       END_IF;
                   END_REGION
               #S119_BW_LOAD_UNLOAD_SEQ_ERROR:
                   REGION S119_BW_LOAD_UNLOAD_SEQ_ERROR
                       IF #sInterface.SequenceReleased AND "AlwaysTRUE" THEN
                           #sCurrent_Step_NB := #S999_ERROR;
                           #sCheck_Step_Condition := FALSE;
                       END_IF;
                   END_REGION

               #S120_PARTS_CTRL_OUT_SEQ_REQUEST:
                   REGION S120_PARTS_CTRL_OUT_SEQ_REQUEST
                       IF #sInterface.SequenceReleased AND #ioControlOutSeq.SequenceRun THEN
                           #sCurrent_Step_NB := #S122_PARTS_CTRL_OUT_SEQ_IN_PROGRESS;
                           #sCheck_Step_Condition := FALSE;
                       ELSIF #sInterface.SequenceReleased AND #ioControlOutSeq.Error THEN
                           #sCurrent_Step_NB := #S129_PARTS_CTRL_OUT_SEQ_ERROR;
                           #sCheck_Step_Condition := FALSE;
                       END_IF;
                   END_REGION
               #S122_PARTS_CTRL_OUT_SEQ_IN_PROGRESS:
                   REGION S122_PARTS_CTRL_OUT_SEQ_IN_PROGRESS
                       IF #sInterface.SequenceReleased AND #ioControlOutSeq.JobDone THEN
                           #sCurrent_Step_NB := #S124_PARTS_CTRL_OUT_SEQ_ACQUIT;
                           #sCheck_Step_Condition := FALSE;
                       ELSIF #sInterface.SequenceReleased AND #ioControlOutSeq.Error THEN
                           #sCurrent_Step_NB := #S129_PARTS_CTRL_OUT_SEQ_ERROR;
                           #sCheck_Step_Condition := FALSE;
                       END_IF;
                   END_REGION
               #S124_PARTS_CTRL_OUT_SEQ_ACQUIT:
                   REGION S124_PARTS_CTRL_OUT_SEQ_ACQUIT
                       IF #sInterface.SequenceReleased AND #iPartCtrlOutOK AND NOT #iPartCtrlOutNOK THEN
                           #sCurrent_Step_NB := #S130_CHECK_CYCLE_STOP;
                           #sCheck_Step_Condition := FALSE;
                       ELSIF #sInterface.SequenceReleased AND NOT #iPartCtrlOutOK AND #iPartCtrlOutNOK THEN
                           #sCurrent_Step_NB := #S310_ACT_PART_CTRL_OUT_SEQ_REQUEST;
                           #sCheck_Step_Condition := FALSE;
                       END_IF;
                   END_REGION
               #S129_PARTS_CTRL_OUT_SEQ_ERROR:
                   REGION S129_PARTS_CTRL_OUT_SEQ_ERROR
                       IF #sInterface.SequenceReleased AND "AlwaysTRUE" THEN
                           #sCurrent_Step_NB := #S999_ERROR;
                           #sCheck_Step_Condition := FALSE;
                       END_IF;
                   END_REGION

               #S130_CHECK_CYCLE_STOP:
                   REGION S130_CHECK_CYCLE_STOP
                       IF #sInterface.SequenceReleased AND #iJobReq THEN
                           #sCurrent_Step_NB := #S20_EXT_LOAD_UNLOAD_SEQ_REQUEST;
                           #sCheck_Step_Condition := FALSE;
                       ELSIF #sInterface.SequenceReleased AND NOT #iJobReq THEN
                           #sCurrent_Step_NB := #S140_EXT_LOAD_UNLOAD_SEQ_REQUEST;
                           #sCheck_Step_Condition := FALSE;
                       END_IF;
                   END_REGION

               #S140_EXT_LOAD_UNLOAD_SEQ_REQUEST:
                   REGION S140_EXT_LOAD_UNLOAD_SEQ_REQUEST
                       IF #sInterface.SequenceReleased AND #ioExtLoadUnloadSeq.SequenceRun THEN
                           #sCurrent_Step_NB := #S142_EXT_LOAD_UNLOAD_SEQ_IN_PROGRESS;
                           #sCheck_Step_Condition := FALSE;
                       ELSIF #sInterface.SequenceReleased AND #ioExtLoadUnloadSeq.Error THEN
                           #sCurrent_Step_NB := #S149_EXT_LOAD_UNLOAD_SEQ_ERROR;
                           #sCheck_Step_Condition := FALSE;
                       END_IF;
                   END_REGION
               #S142_EXT_LOAD_UNLOAD_SEQ_IN_PROGRESS:
                   REGION S142_EXT_LOAD_UNLOAD_SEQ_IN_PROGRESS
                       IF #sInterface.SequenceReleased AND #ioExtLoadUnloadSeq.JobDone THEN
                           #sCurrent_Step_NB := #S144_EXT_LOAD_UNLOAD_SEQ_ACQUIT;
                           #sCheck_Step_Condition := FALSE;
                       ELSIF #sInterface.SequenceReleased AND #ioExtLoadUnloadSeq.Error THEN
                           #sCurrent_Step_NB := #S149_EXT_LOAD_UNLOAD_SEQ_ERROR;
                           #sCheck_Step_Condition := FALSE;
                       END_IF;
                   END_REGION
               #S144_EXT_LOAD_UNLOAD_SEQ_ACQUIT:
                   REGION S144_EXT_LOAD_UNLOAD_SEQ_ACQUIT
                       IF #sInterface.SequenceReleased AND "AlwaysTRUE" THEN
                           #sCurrent_Step_NB := #S00_INIT_STEP;
                           #sCheck_Step_Condition := FALSE;
                       END_IF;
                   END_REGION
               #S149_EXT_LOAD_UNLOAD_SEQ_ERROR:
                   REGION S149_EXT_LOAD_UNLOAD_SEQ_ERROR
                       IF #sInterface.SequenceReleased AND "AlwaysTRUE" THEN
                           #sCurrent_Step_NB := #S999_ERROR;
                           #sCheck_Step_Condition := FALSE;
                       END_IF;
                   END_REGION

               #S200_BLOWING_SEQ_REQUEST:
                   REGION S200_BLOWING_SEQ_REQUEST
                       IF #sInterface.SequenceReleased AND #ioBlowingSeq.SequenceRun THEN
                           #sCurrent_Step_NB := #S202_BLOWING_SEQ_IN_PROGRESS;
                           #sCheck_Step_Condition := FALSE;
                       ELSIF #sInterface.SequenceReleased AND #ioBlowingSeq.Error THEN
                           #sCurrent_Step_NB := #S209_BLOWING_SEQ_ERROR;
                           #sCheck_Step_Condition := FALSE;
                       END_IF;
                   END_REGION
               #S202_BLOWING_SEQ_IN_PROGRESS:
                   REGION S202_BLOWING_SEQ_IN_PROGRESS
                       IF #sInterface.SequenceReleased AND #ioBlowingSeq.JobDone THEN
                           #sCurrent_Step_NB := #S204_BLOWING_SEQ_ACQUIT;
                           #sCheck_Step_Condition := FALSE;
                       ELSIF #sInterface.SequenceReleased AND #ioBlowingSeq.Error THEN
                           #sCurrent_Step_NB := #S209_BLOWING_SEQ_ERROR;
                           #sCheck_Step_Condition := FALSE;
                       END_IF;
                   END_REGION
               #S204_BLOWING_SEQ_ACQUIT:
                   REGION S204_BLOWING_SEQ_ACQUIT
                       IF #sInterface.SequenceReleased AND NOT #iOnePieceMode THEN
                           #sCurrent_Step_NB := #S80_INT_LOAD_UNLOAD_SEQ_REQUEST;
                           #sCheck_Step_Condition := FALSE;
                       ELSIF #sInterface.SequenceReleased AND #iOnePieceMode THEN
                           #sCurrent_Step_NB := #S210_INT_LOAD_UNLOAD_OP_SEQ_REQUEST;
                           #sCheck_Step_Condition := FALSE;
                       END_IF;
                   END_REGION
               #S209_BLOWING_SEQ_ERROR:
                   REGION S209_BLOWING_SEQ_ERROR
                       IF #sInterface.SequenceReleased AND "AlwaysTRUE" THEN
                           #sCurrent_Step_NB := #S999_ERROR;
                           #sCheck_Step_Condition := FALSE;
                       END_IF;
                   END_REGION

               #S210_INT_LOAD_UNLOAD_OP_SEQ_REQUEST:
                   REGION S210_INT_LOAD_UNLOAD_OP_SEQ_REQUEST
                       IF #sInterface.SequenceReleased AND #ioIntLoadUnloadOP_Seq.SequenceRun THEN
                           #sCurrent_Step_NB := #S212_INT_LOAD_UNLOAD_OP_SEQ_IN_PROGRESS;
                           #sCheck_Step_Condition := FALSE;
                       ELSIF #sInterface.SequenceReleased AND #ioIntLoadUnloadOP_Seq.Error THEN
                           #sCurrent_Step_NB := #S219_INT_LOAD_UNLOAD_OP_SEQ_ERROR;
                           #sCheck_Step_Condition := FALSE;
                       END_IF;
                   END_REGION
               #S212_INT_LOAD_UNLOAD_OP_SEQ_IN_PROGRESS:
                   REGION S212_INT_LOAD_UNLOAD_OP_SEQ_IN_PROGRESS
                       IF #sInterface.SequenceReleased AND #ioIntLoadUnloadOP_Seq.JobDone THEN
                           #sCurrent_Step_NB := #S214_INT_LOAD_UNLOAD_OP_SEQ_ACQUIT;
                           #sCheck_Step_Condition := FALSE;
                       ELSIF #sInterface.SequenceReleased AND #ioIntLoadUnloadOP_Seq.Error THEN
                           #sCurrent_Step_NB := #S219_INT_LOAD_UNLOAD_OP_SEQ_ERROR;
                           #sCheck_Step_Condition := FALSE;
                       END_IF;
                   END_REGION
               #S214_INT_LOAD_UNLOAD_OP_SEQ_ACQUIT:
                   REGION S214_INT_LOAD_UNLOAD_OP_SEQ_ACQUIT
                       IF #sInterface.SequenceReleased AND "AlwaysTRUE" THEN
                           #sCurrent_Step_NB := #S90_TRANSFER_V_AND_W_AXIS_TO_NC;
                           #sCheck_Step_Condition := FALSE;
                       END_IF;
                   END_REGION
               #S219_INT_LOAD_UNLOAD_OP_SEQ_ERROR:
                   REGION S219_INT_LOAD_UNLOAD_OP_SEQ_ERROR
                       IF #sInterface.SequenceReleased AND "AlwaysTRUE" THEN
                           #sCurrent_Step_NB := #S999_ERROR;
                           #sCheck_Step_Condition := FALSE;
                       END_IF;
                   END_REGION

               #S300_ACT_PART_CTRL_IN_SEQ_REQUEST:
                   REGION S300_ACT_PART_CTRL_IN_SEQ_REQUEST
                       IF #sInterface.SequenceReleased AND #ioActPartControlInSeq.SequenceRun THEN
                           #sCurrent_Step_NB := #S302_ACT_PART_CTRL_IN_SEQ_IN_PROGRESS;
                           #sCheck_Step_Condition := FALSE;
                       ELSIF #sInterface.SequenceReleased AND #ioActPartControlInSeq.Error THEN
                           #sCurrent_Step_NB := #S309_ACT_PART_CTRL_IN_SEQ_ERROR;
                           #sCheck_Step_Condition := FALSE;
                       END_IF;
                   END_REGION
               #S302_ACT_PART_CTRL_IN_SEQ_IN_PROGRESS:
                   REGION S302_ACT_PART_CTRL_IN_SEQ_IN_PROGRESS
                       IF #sInterface.SequenceReleased AND #ioActPartControlInSeq.JobDone THEN
                           #sCurrent_Step_NB := #S304_ACT_PART_CTRL_IN_SEQ_ACQUIT;
                           #sCheck_Step_Condition := FALSE;
                       ELSIF #sInterface.SequenceReleased AND #ioActPartControlInSeq.Error THEN
                           #sCurrent_Step_NB := #S309_ACT_PART_CTRL_IN_SEQ_ERROR;
                           #sCheck_Step_Condition := FALSE;
                       END_IF;
                   END_REGION
               #S304_ACT_PART_CTRL_IN_SEQ_ACQUIT:
                   REGION S304_ACT_PART_CTRL_IN_SEQ_ACQUIT
                       IF #sInterface.SequenceReleased AND #iPartCtrlInContinuationStep THEN
                           #sCurrent_Step_NB := #S40_BW_LOAD_UNLOAD_SEQ_REQUEST;
                           #sCheck_Step_Condition := FALSE;
                       ELSIF #sInterface.SequenceReleased AND #iPartCtrlInRestartStep THEN
                           #sCurrent_Step_NB := #S30_PARTS_CTRL_IN_SEQ_REQUEST;
                           #sCheck_Step_Condition := FALSE;
                       END_IF;
                   END_REGION
               #S309_ACT_PART_CTRL_IN_SEQ_ERROR:
                   REGION S309_ACT_PART_CTRL_IN_SEQ_ERROR
                       IF #sInterface.SequenceReleased AND "AlwaysTRUE" THEN
                           #sCurrent_Step_NB := #S999_ERROR;
                           #sCheck_Step_Condition := FALSE;
                       END_IF;
                   END_REGION

               #S310_ACT_PART_CTRL_OUT_SEQ_REQUEST:
                   REGION S310_ACT_PART_CTRL_OUT_SEQ_REQUEST
                       IF #sInterface.SequenceReleased AND #ioActPartControlOutSeq.SequenceRun THEN
                           #sCurrent_Step_NB := #S312_ACT_PART_CTRL_OUT_SEQ_IN_PROGRESS;
                           #sCheck_Step_Condition := FALSE;
                       ELSIF #sInterface.SequenceReleased AND #ioActPartControlOutSeq.Error THEN
                           #sCurrent_Step_NB := #S319_ACT_PART_CTRL_OUT_SEQ_ERROR;
                           #sCheck_Step_Condition := FALSE;
                       END_IF;
                   END_REGION
               #S312_ACT_PART_CTRL_OUT_SEQ_IN_PROGRESS:
                   REGION S312_ACT_PART_CTRL_OUT_SEQ_IN_PROGRESS
                       IF #sInterface.SequenceReleased AND #ioActPartControlOutSeq.JobDone THEN
                           #sCurrent_Step_NB := #S314_ACT_PART_CTRL_OUT_SEQ_ACQUIT;
                           #sCheck_Step_Condition := FALSE;
                       ELSIF #sInterface.SequenceReleased AND #ioActPartControlOutSeq.Error THEN
                           #sCurrent_Step_NB := #S319_ACT_PART_CTRL_OUT_SEQ_ERROR;
                           #sCheck_Step_Condition := FALSE;
                       END_IF;
                   END_REGION
               #S314_ACT_PART_CTRL_OUT_SEQ_ACQUIT:
                   REGION S314_ACT_PART_CTRL_OUT_SEQ_ACQUIT
                       IF #sInterface.SequenceReleased AND #iPartCtrlOutContinuationStep THEN
                           #sCurrent_Step_NB := #S130_CHECK_CYCLE_STOP;
                           #sCheck_Step_Condition := FALSE;
                       ELSIF #sInterface.SequenceReleased AND #iPartCtrlOutRestartStep THEN
                           #sCurrent_Step_NB := #S120_PARTS_CTRL_OUT_SEQ_REQUEST;
                           #sCheck_Step_Condition := FALSE;
                       END_IF;
                   END_REGION
               #S319_ACT_PART_CTRL_OUT_SEQ_ERROR:
                   REGION S319_ACT_PART_CTRL_OUT_SEQ_ERROR
                       IF #sInterface.SequenceReleased AND "AlwaysTRUE" THEN
                           #sCurrent_Step_NB := #S999_ERROR;
                           #sCheck_Step_Condition := FALSE;
                       END_IF;
                   END_REGION

               #S320_ACT_BW_CTRL_IN_SEQ_REQUEST:
                   REGION S320_ACT_BW_CTRL_IN_SEQ_REQUEST
                       IF #sInterface.SequenceReleased AND #ioActBwControlInSeq.SequenceRun THEN
                           #sCurrent_Step_NB := #S322_ACT_BW_CTRL_IN_SEQ_IN_PROGRESS;
                           #sCheck_Step_Condition := FALSE;
                       ELSIF #sInterface.SequenceReleased AND #ioActBwControlInSeq.Error THEN
                           #sCurrent_Step_NB := #S329_ACT_BW_CTRL_IN_SEQ_ERROR;
                           #sCheck_Step_Condition := FALSE;
                       END_IF;
                   END_REGION
               #S322_ACT_BW_CTRL_IN_SEQ_IN_PROGRESS:
                   REGION S322_ACT_BW_CTRL_IN_SEQ_IN_PROGRESS
                       IF #sInterface.SequenceReleased AND #ioActBwControlInSeq.JobDone THEN
                           #sCurrent_Step_NB := #S324_ACT_BW_CTRL_IN_SEQ_ACQUIT;
                           #sCheck_Step_Condition := FALSE;
                       ELSIF #sInterface.SequenceReleased AND #ioActBwControlInSeq.Error THEN
                           #sCurrent_Step_NB := #S329_ACT_BW_CTRL_IN_SEQ_ERROR;
                           #sCheck_Step_Condition := FALSE;
                       END_IF;
                   END_REGION
               #S324_ACT_BW_CTRL_IN_SEQ_ACQUIT:
                   REGION S324_ACT_BW_CTRL_IN_SEQ_ACQUIT
                       IF #sInterface.SequenceReleased AND #iBwCtrlInContinuationStep THEN
                           #sCurrent_Step_NB := #S60_SHUTTLE_INT_SEQ_REQUEST;
                           #sCheck_Step_Condition := FALSE;
                       ELSIF #sInterface.SequenceReleased AND #iBwCtrlInRestartStep THEN
                           #sCurrent_Step_NB := #S40_BW_LOAD_UNLOAD_SEQ_REQUEST;
                           #sCheck_Step_Condition := FALSE;
                       END_IF;
                   END_REGION
               #S329_ACT_BW_CTRL_IN_SEQ_ERROR:
                   REGION S329_ACT_BW_CTRL_IN_SEQ_ERROR
                       IF #sInterface.SequenceReleased AND "AlwaysTRUE" THEN
                           #sCurrent_Step_NB := #S999_ERROR;
                           #sCheck_Step_Condition := FALSE;
                       END_IF;
                   END_REGION

               #S999_ERROR:
                   REGION S999_ERROR
                       IF #sInterface.SequenceReleased AND "AlwaysFALSE" THEN
                           #sCurrent_Step_NB := #S999_ERROR;
                           #sCheck_Step_Condition := FALSE;
                       END_IF;
                   END_REGION
               ELSE
                   #sInterface.Error := TRUE;
           END_CASE;
       END_IF;
   END_REGION

   REGION Outputs Update
       #oGripperAxisRequest := #sGripperAxisRequest;
       #oGripperAxisRelease := #sGripperAxisRelease;
   END_REGION

   REGION Steps - Date and Time History
       IF #sHistory.Activation THEN
           IF #sHistory.Steps[0] <> #sCurrent_Step_NB THEN
               FOR #tIndex := 98 TO 0 BY -1 DO
                   #sHistory.Steps[#tIndex + 1] := #sHistory.Steps[#tIndex];
                   #sHistory.Date_Time[#tIndex + 1] := #sHistory.Date_Time[#tIndex];
               END_FOR;
               #sHistory.Steps[0] := #sCurrent_Step_NB;
               #sHistory.Date_Time[0] := #iPLC_DateAndTime;
           END_IF;
       END_IF;
   END_REGION

   REGION Steps Text
       #StepText(iErrorCode := #sCurrent_Step_NB,
                 oErrorText => #StepText.oErrorText);
   END_REGION
END_FUNCTION_BLOCK

FUNCTION_BLOCK "FB_GetTextErrorCode"   // FB301, SCL
{ S7_Optimized_Access := 'TRUE' }
// stored: AutoNumber false, MemoryReserve 100, SetENOAutomatically false
   VAR_INPUT
      iErrorCode { ExternalAccessible := 'False'; ExternalVisible := 'False'; ExternalWritable := 'False'} : Int;
   END_VAR
   VAR_OUTPUT
      oErrorText { ExternalAccessible := 'False'; ExternalVisible := 'False'; ExternalWritable := 'False'} : String;
   END_VAR
   VAR RETAIN
      sCode_error : Array[0..100] of Struct
         ErrorCode : Int;
         ErrorText : String[64];
      END_STRUCT;
   END_VAR
   VAR_TEMP
      tIndex : Int;
   END_VAR
   // sCode_error[0].ErrorCode := 0;
   // sCode_error[1].ErrorCode := 9999;
   // sCode_error[2].ErrorCode := 7504;
   // sCode_error[3].ErrorCode := 8000;
   // sCode_error[4].ErrorCode := 7064;
   // sCode_error[5].ErrorCode := 7004;
   // sCode_error[6].ErrorCode := 27564;
   // sCode_error[7].ErrorCode := 7068;
   // sCode_error[8].ErrorCode := 17504;
   // sCode_error[9].ErrorCode := 6564;
   // sCode_error[10].ErrorCode := 9064;
   // sCode_error[11].ErrorCode := 9004;
   // sCode_error[12].ErrorCode := 9010;
   // sCode_error[13..100].ErrorCode := 0;
   // sCode_error[0].ErrorText := 'Unknown, No text';
   // sCode_error[1].ErrorText := 'Part start drilling, but not finished';
   // sCode_error[2].ErrorText := 'woz out of tolerance';
   // sCode_error[3].ErrorText := 'runout';
   // sCode_error[4].ErrorText := 'Z out of range';
   // sCode_error[5].ErrorText := 'Z out of tolerance';
   // sCode_error[6].ErrorText := 'woz out of range';
   // sCode_error[7].ErrorText := 'z out of range and tolerance';
   // sCode_error[8].ErrorText := 'part not clamped';
   // sCode_error[9].ErrorText := 'Woc';
   // sCode_error[10..11].ErrorText := 'Drilled part with broken BW';
   // sCode_error[12].ErrorText := 'Drilled part with N2 not enough';
   // sCode_error[13..100].ErrorText := '';
BEGIN
       //==================================================================================
       // POSALUX Swiss SA / (C) Copyright 2025
       //----------------------------------------------------------------------------------
       // Title: Power de la machine
       // Comment/Function: Generates an error text based on an error number
       //           If the Error code is not found, "ErrorCode: Code unknow" is displayed          
       // Author: Fabien WALDT
       // Engineering: TIA Portal v17
       //----------------------------------------------------------------------------------
       // Change log table:
       // Version  | Date     | Expert in charge | Changes applied
       // ---------|----------|------------------|------------------------------------
       // 00.00.01 | 20250415 | WFA              | First released version
       // ==================================================================================
       REGION NO Error
           IF #iErrorCode = 0 THEN
               #oErrorText := #sCode_error[0].ErrorText;
           END_IF;
       END_REGION

       REGION Error
           IF #iErrorCode > 0 THEN
               FOR #tIndex := 1 TO 100 DO
                   IF #iErrorCode = #sCode_error[#tIndex].ErrorCode THEN
                       // Error text found in the list
                       #oErrorText := #sCode_error[#tIndex].ErrorText;
                       EXIT;
                   END_IF;
                   // Error text not found in the list
                   #oErrorText := CONCAT(IN1 := DELETE(IN := INT_TO_STRING(#iErrorCode), L := 1, P := 1), IN2 := ': Code unknow');
               END_FOR;
           END_IF;
       END_REGION
END_FUNCTION_BLOCK

